RoboDK station: kr30 cnc 040719 6.rdk

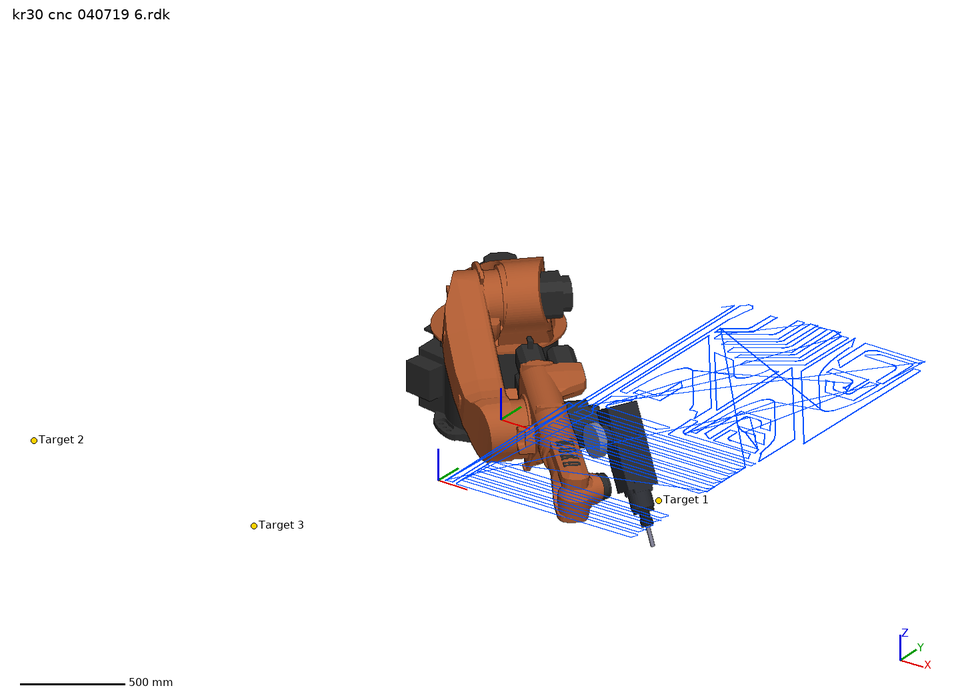
[picture v0: the station drawn from its stored meshes, robots at their saved joint values, targets as dots, program paths as lines]
Station kr30 cnc 040719 6. Poses are relative to the parent item; angles as X-Y-Z fixed-axis rotations.
  - frame KUKA KR 30 HA Base at (0, 0, 0) mm
    - robot KUKA KR 30 HA: 6 axes, payload 30 kg, reach 2033 mm, repeatability 0.05 mm, weight 665 kg
        modified DH rows (alpha deg, a mm, theta deg, d mm): 0, 0, 0, 815; -90, 350, 0, 0; 0, 850, -90, 0; -90, 145, 0, 820; 90, 0, 0, 0; -90, 0, 180, 170
        joint limits [-185, -135, -120, -350, -119, -350] to [185, 35, 158, 350, 119, 350]; home [0, -90, 90, 0, 0, 0]; saved at [44.88, 20.858, -14.182, 92.407, -109.74, -52.906]
      - tool 1/2" End Mill TCP, TCP at (337.71, -2.2, 160.57) mm, size 692.9 x 170 x 256 mm
    - frame Reference Rhino at (451.13, -1162.89, 269.68) mm
      - target Target 1 (Cartesian target) at (994.45, 406.4, 10) mm, rotated rx 0 ry 90 rz -60.43 deg; joints [16.304, -19.243, 71.371, -50.859, -63.853, 28.433] of KUKA KR 30 HA
      - target Target 2 (Cartesian target) at (-1810.84, -765.32, 10.08) mm, rotated rx 49.23 ry 89.99 rz -110.09 deg; joints [109.009, -5.295, 40.673, -64.339, -58.629, 47.297] of KUKA KR 30 HA
      - target Target 3 (Cartesian target) at (-425.52, -920.6, 10.08) mm, rotated rx 49.23 ry 89.99 rz -69.31 deg; joints [71.775, -8.447, 47.414, -59.408, -57.827, 42.008] of KUKA KR 30 HA
      - object RhinoPart at (0, 0, 0) mm
  - machining project RhinoPart Settings: C:/Users/Julian Ramirez.DESKTOP-JVDE542/Desktop/ELMER SHEET 1 TEST 3.nc | rotX(0) | rotY(270)*rotX(-65)
  - object box at (500, 500, 500) mm, size 250 x 250 x 250 mm, geometry from box.sld
  - program RhinoPart (634 instructions, listed below)
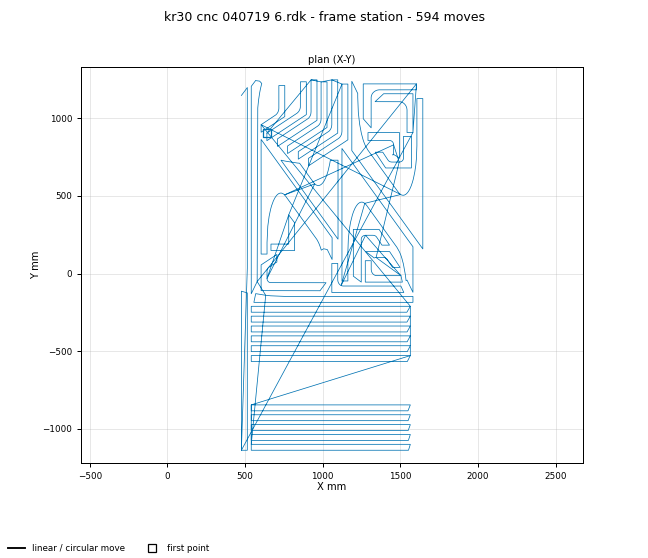
[picture p0: tool path of kr30 cnc 040719 6.rdk in frame station, 594 of 594 moves have a stored position in this frame; points joined in program order, loops and branches not executed]

--- program RhinoPart (robot KUKA KR 30 HA) ---
  Smooth(1)
  Set Ref.: Reference Rhino
  Set Tool: 1/2" End Mill TCP
  Show 1/2" End Mill TCP
  Set speed (2000.0 mm/s)
  MoveJ 1 to (189.6, 2067.69, 0) mm, rotated rx 0 ry 90 rz 65 deg; joints [-50.535, -45.887, 156.75, 15.433, -110.173, 5.438]
  MoveL 2 to (189.6, 2067.69, 0) mm, rotated rx 0 ry 90 rz 65 deg; joints [-50.535, -45.887, 156.75, 15.433, -110.173, 5.438]
  MoveL 3 to (189.6, 2067.69, 0) mm, rotated rx 0 ry 90 rz 65 deg; joints [-50.535, -45.887, 156.75, 15.433, -110.173, 5.438]
  Set speed (60.0 mm/s)
  MoveL 4 to (189.6, 2019.15, 0) mm, rotated rx 90 ry 80 rz 155 deg; joints [-43.975, -44.854, 157.735, 22.646, -111.28, -1.39]
  MoveL 5 to (443.6, 2187.03, 0) mm, rotated rx 0 ry 90 rz 65 deg; joints [-43.932, -46.602, 138.926, 21.084, -92.169, 0.836]
  MoveL 6 to (443.6, 2398.44, 0) mm, rotated rx 0 ry 90 rz 65 deg; joints [-51.209, -43.939, 127.221, 13.883, -83.477, -1.608]
  MoveL 7 to (405.5, 2398.44, 0) mm, rotated rx 0 ry 90 rz 65 deg; joints [-52.653, -44.436, 129.033, 12.401, -84.722, -1.159]
  MoveL 8 to (405.5, 2241.51, 0) mm, rotated rx 0 ry 90 rz 65 deg; joints [-47.49, -46.452, 138.026, 17.516, -91.501, 0.474]
  MoveL 9 to (405.1, 2234.61, 0) mm, rotated rx 0 ry 90 rz 65 deg; joints [-47.252, -46.518, 138.415, 17.757, -91.807, 0.578]
  MoveL 10 to (403.91, 2227.8, 0) mm, rotated rx 0 ry 90 rz 65 deg; joints [-47.047, -46.587, 138.835, 17.966, -92.138, 0.693]
  MoveL 11 to (401.94, 2221.18, 0) mm, rotated rx 0 ry 90 rz 65 deg; joints [-46.878, -46.658, 139.282, 18.139, -92.494, 0.817]
  MoveL 12 to (399.2, 2214.83, 0) mm, rotated rx 0 ry 90 rz 65 deg; joints [-46.749, -46.729, 139.751, 18.275, -92.87, 0.947]
  MoveL 13 to (395.69, 2208.84, 0) mm, rotated rx 0 ry 90 rz 65 deg; joints [-46.662, -46.8, 140.238, 18.369, -93.264, 1.083]
  MoveL 14 to (391.47, 2203.34, 0) mm, rotated rx 0 ry 90 rz 65 deg; joints [-46.623, -46.867, 140.732, 18.416, -93.667, 1.22]
  MoveL 15 to (386.58, 2198.44, 0) mm, rotated rx 0 ry 90 rz 65 deg; joints [-46.634, -46.931, 141.227, 18.415, -94.076, 1.356]
  MoveL 16 to (383.89, 2196.24, 0) mm, rotated rx 0 ry 90 rz 65 deg; joints [-46.659, -46.962, 141.472, 18.394, -94.281, 1.422]
  MoveL 17 to (381.06, 2194.23, 0) mm, rotated rx 0 ry 90 rz 65 deg; joints [-46.697, -46.991, 141.716, 18.361, -94.486, 1.487]
  MoveL 18 to (189.6, 2067.69, 0) mm, rotated rx 0 ry 90 rz 65 deg; joints [-50.535, -45.887, 156.75, 15.433, -110.173, 5.438]
  MoveL 19 to (474.07, 2410.87, 0) mm, rotated rx 0 ry 90 rz 65 deg; joints [-50.466, -43.286, 124.966, 14.682, -81.949, -2.102]
  Set speed (60.0 mm/s)
  MoveL 20 to (512.17, 2410.87, 0) mm, rotated rx 0 ry 90 rz 65 deg; joints [-49.125, -42.694, 123.02, 16.093, -80.698, -2.67]
  MoveL 21 to (512.17, 2150.2, 0) mm, rotated rx 0 ry 90 rz 65 deg; joints [-39.968, -46.268, 137.006, 25.034, -90.668, 0.312]
  MoveL 22 to (258.17, 1982.32, 0) mm, rotated rx 0 ry 90 rz 65 deg; joints [-42.535, -45.52, 157.698, 24.062, -110.416, 8.854]
  MoveL 23 to (258.17, 2030.85, 0) mm, rotated rx 0 ry 90 rz 65 deg; joints [-45.085, -46.283, 155.538, 20.995, -108.063, 6.786]
  MoveL 24 to (449.63, 2157.39, 0) mm, rotated rx 0 ry 90 rz 65 deg; joints [-42.511, -46.776, 140.073, 22.522, -93.046, 1.262]
  MoveL 25 to (455.15, 2161.61, 0) mm, rotated rx 0 ry 90 rz 65 deg; joints [-42.477, -46.703, 139.574, 22.548, -92.652, 1.101]
  MoveL 26 to (460.04, 2166.51, 0) mm, rotated rx 0 ry 90 rz 65 deg; joints [-42.494, -46.625, 139.075, 22.524, -92.263, 0.938]
  MoveL 27 to (464.26, 2172, 0) mm, rotated rx 0 ry 90 rz 65 deg; joints [-42.56, -46.545, 138.581, 22.453, -91.882, 0.777]
  MoveL 28 to (467.77, 2178, 0) mm, rotated rx 0 ry 90 rz 65 deg; joints [-42.67, -46.464, 138.099, 22.338, -91.512, 0.621]
  MoveL 29 to (470.51, 2184.35, 0) mm, rotated rx 0 ry 90 rz 65 deg; joints [-42.822, -46.384, 137.638, 22.183, -91.162, 0.474]
  MoveL 30 to (472.48, 2190.97, 0) mm, rotated rx 0 ry 90 rz 65 deg; joints [-43.01, -46.305, 137.204, 21.992, -90.834, 0.337]
  MoveL 31 to (474.07, 2204.68, 0) mm, rotated rx 0 ry 90 rz 65 deg; joints [-43.485, -46.159, 136.432, 21.516, -90.253, 0.1]
  MoveL 32 to (474.07, 2410.87, 0) mm, rotated rx 0 ry 90 rz 65 deg; joints [-50.466, -43.286, 124.966, 14.682, -81.949, -2.102]
  MoveL 33 to (538.73, 2397.73, 0) mm, rotated rx 0 ry 90 rz 65 deg; joints [-47.823, -42.501, 122.4, 17.431, -80.354, -3.011]
  Set speed (60.0 mm/s)
  MoveL 34 to (538.73, 2158.69, 0) mm, rotated rx 0 ry 90 rz 65 deg; joints [-39.418, -45.892, 135.103, 25.584, -89.288, -0.341]
  MoveL 35 to (537.14, 2144.98, 0) mm, rotated rx 0 ry 90 rz 65 deg; joints [-38.913, -46.041, 135.833, 26.087, -89.813, -0.092]
  MoveL 36 to (535.17, 2138.36, 0) mm, rotated rx 0 ry 90 rz 65 deg; joints [-38.706, -46.124, 136.251, 26.294, -90.114, 0.056]
  MoveL 37 to (532.43, 2132.01, 0) mm, rotated rx 0 ry 90 rz 65 deg; joints [-38.533, -46.211, 136.699, 26.467, -90.437, 0.218]
  MoveL 38 to (528.92, 2126.02, 0) mm, rotated rx 0 ry 90 rz 65 deg; joints [-38.399, -46.299, 137.173, 26.603, -90.782, 0.391]
  MoveL 39 to (524.7, 2120.53, 0) mm, rotated rx 0 ry 90 rz 65 deg; joints [-38.309, -46.388, 137.664, 26.697, -91.14, 0.573]
  MoveL 40 to (519.81, 2115.63, 0) mm, rotated rx 0 ry 90 rz 65 deg; joints [-38.264, -46.475, 138.164, 26.746, -91.508, 0.76]
  MoveL 41 to (514.29, 2111.41, 0) mm, rotated rx 0 ry 90 rz 65 deg; joints [-38.27, -46.56, 138.668, 26.745, -91.883, 0.949]
  MoveL 42 to (322.83, 1984.87, 0) mm, rotated rx 0 ry 90 rz 65 deg; joints [-39.614, -46.576, 154.441, 26.5, -106.091, 7.868]
  MoveL 43 to (322.83, 1936.34, 0) mm, rotated rx 0 ry 90 rz 65 deg; joints [-36.903, -46.012, 156.394, 29.663, -107.892, 9.925]
  MoveL 44 to (576.83, 2104.21, 0) mm, rotated rx 0 ry 90 rz 65 deg; joints [-35.947, -45.94, 135.336, 29.055, -89.472, -0.293]
  MoveL 45 to (576.83, 2397.73, 0) mm, rotated rx 0 ry 90 rz 65 deg; joints [-46.568, -41.834, 120.316, 18.784, -79.08, -3.686]
  MoveL 46 to (538.73, 2397.73, 0) mm, rotated rx 0 ry 90 rz 65 deg; joints [-47.823, -42.501, 122.4, 17.431, -80.354, -3.011]
  MoveL 47 to (607.72, 2410.87, 0) mm, rotated rx 0 ry 90 rz 65 deg; joints [-45.987, -40.997, 117.795, 19.491, -77.53, -4.37]
  Set speed (60.0 mm/s)
  MoveL 48 to (645.82, 2410.87, 0) mm, rotated rx 0 ry 90 rz 65 deg; joints [-44.821, -40.232, 115.572, 20.801, -76.258, -5.156]
  MoveL 49 to (645.82, 2068.09, 0) mm, rotated rx 0 ry 90 rz 65 deg; joints [-32.413, -45.334, 132.596, 32.617, -87.693, -1.476]
  MoveL 50 to (391.82, 1900.22, 0) mm, rotated rx 0 ry 90 rz 65 deg; joints [-32.027, -46.673, 154.021, 34.202, -104.486, 9.648]
  MoveL 51 to (391.82, 1948.75, 0) mm, rotated rx 0 ry 90 rz 65 deg; joints [-34.789, -47.001, 152.253, 31.112, -103.14, 7.812]
  MoveL 52 to (583.27, 2075.29, 0) mm, rotated rx 0 ry 90 rz 65 deg; joints [-34.508, -46.11, 136.177, 30.492, -90.058, 0.034]
  MoveL 53 to (588.8, 2079.51, 0) mm, rotated rx 0 ry 90 rz 65 deg; joints [-34.526, -46.008, 135.666, 30.474, -89.706, -0.173]
  MoveL 54 to (593.69, 2084.41, 0) mm, rotated rx 0 ry 90 rz 65 deg; joints [-34.592, -45.905, 135.164, 30.41, -89.361, -0.375]
  MoveL 55 to (597.91, 2089.9, 0) mm, rotated rx 0 ry 90 rz 65 deg; joints [-34.703, -45.802, 134.676, 30.302, -89.028, -0.568]
  MoveL 56 to (601.42, 2095.89, 0) mm, rotated rx 0 ry 90 rz 65 deg; joints [-34.854, -45.7, 134.208, 30.155, -88.709, -0.75]
  MoveL 57 to (604.16, 2102.24, 0) mm, rotated rx 0 ry 90 rz 65 deg; joints [-35.041, -45.603, 133.769, 29.972, -88.411, -0.916]
  MoveL 58 to (606.13, 2108.87, 0) mm, rotated rx 0 ry 90 rz 65 deg; joints [-35.26, -45.512, 133.364, 29.757, -88.135, -1.066]
  MoveL 59 to (607.72, 2122.58, 0) mm, rotated rx 0 ry 90 rz 65 deg; joints [-35.781, -45.352, 132.671, 29.246, -87.661, -1.309]
  MoveL 60 to (607.72, 2410.87, 0) mm, rotated rx 0 ry 90 rz 65 deg; joints [-45.987, -40.997, 117.795, 19.491, -77.53, -4.37]
  MoveL 61 to (673.1, 2383.75, 0) mm, rotated rx 0 ry 90 rz 65 deg; joints [-43.185, -40.209, 115.506, 22.481, -76.371, -5.569]
  Set speed (60.0 mm/s)
  MoveL 62 to (673.1, 2079.03, 0) mm, rotated rx 0 ry 90 rz 65 deg; joints [-32.147, -44.797, 130.411, 32.93, -86.317, -2.383]
  MoveL 63 to (671.52, 2065.32, 0) mm, rotated rx 0 ry 90 rz 65 deg; joints [-31.612, -44.962, 131.063, 33.449, -86.745, -2.148]
  MoveL 64 to (669.55, 2058.7, 0) mm, rotated rx 0 ry 90 rz 65 deg; joints [-31.381, -45.058, 131.452, 33.671, -86.997, -1.999]
  MoveL 65 to (666.8, 2052.35, 0) mm, rotated rx 0 ry 90 rz 65 deg; joints [-31.181, -45.163, 131.878, 33.863, -87.272, -1.83]
  MoveL 66 to (663.29, 2046.36, 0) mm, rotated rx 0 ry 90 rz 65 deg; joints [-31.014, -45.273, 132.337, 34.021, -87.566, -1.642]
  MoveL 67 to (659.07, 2040.86, 0) mm, rotated rx 0 ry 90 rz 65 deg; joints [-30.885, -45.387, 132.821, 34.141, -87.876, -1.44]
  MoveL 68 to (654.18, 2035.96, 0) mm, rotated rx 0 ry 90 rz 65 deg; joints [-30.799, -45.503, 133.323, 34.221, -88.198, -1.225]
  MoveL 69 to (648.66, 2031.74, 0) mm, rotated rx 0 ry 90 rz 65 deg; joints [-30.758, -45.619, 133.839, 34.255, -88.528, -1.002]
  MoveL 70 to (457.2, 1905.21, 0) mm, rotated rx 0 ry 90 rz 65 deg; joints [-30.057, -47.242, 150.114, 35.63, -100.522, 7.457]
  MoveL 71 to (457.2, 1856.67, 0) mm, rotated rx 0 ry 90 rz 65 deg; joints [-27.266, -47.081, 151.68, 38.648, -101.498, 9.056]
  MoveL 72 to (711.2, 2024.55, 0) mm, rotated rx 0 ry 90 rz 65 deg; joints [-28.881, -44.696, 130.018, 36.21, -86.223, -2.761]
  MoveL 73 to (711.2, 2383.75, 0) mm, rotated rx 0 ry 90 rz 65 deg; joints [-42.099, -39.37, 113.138, 23.748, -75.078, -6.464]
  MoveL 74 to (673.1, 2383.75, 0) mm, rotated rx 0 ry 90 rz 65 deg; joints [-43.185, -40.209, 115.506, 22.481, -76.371, -5.569]
  MoveL 75 to (330.2, 1541.24, 0) mm, rotated rx 90 ry 60 rz 155 deg; joints [-0.592, -40.922, 154.796, 66.348, -100.068, -8.239]
  Set speed (60.0 mm/s)
  MoveL 76 to (365.54, 1493.75, 0) mm, rotated rx 90 ry 70 rz 155 deg; joints [1.226, -43.408, 156.452, 67.934, -99.079, 1.27]
  MoveL 77 to (368.3, 1490.21, 0) mm, rotated rx 90 ry 70 rz 155 deg; joints [1.481, -43.485, 156.273, 68.137, -98.891, 1.067]
  MoveL 78 to (368.3, 1311.73, 0) mm, rotated rx 90 ry 70 rz 155 deg; joints [14.248, -44.077, 154.711, 79.923, -93.77, 0.302]
  MoveL 79 to (215.9, 1311.73, 0) mm, rotated rx 90 ry 50 rz 155 deg; joints [18.503, -36.104, 155.403, 84.328, -93.174, -10.858]
  MoveL 80 to (215.9, 1353.22, 0) mm, rotated rx 90 ry 50 rz 155 deg; joints [15.495, -35.61, 156.111, 81.791, -94.808, -9.844]
  MoveL 81 to (330.2, 1353.22, 0) mm, rotated rx 90 ry 70 rz 155 deg; joints [11.925, -42.84, 157.646, 78.096, -95.446, 4.238]
  MoveL 82 to (330.2, 1541.24, 0) mm, rotated rx 90 ry 60 rz 155 deg; joints [-0.592, -40.922, 154.796, 66.348, -100.068, -8.239]
  MoveL 83 to (190.5, 1131.98, 0) mm, rotated rx 90 ry 60 rz 155 deg; joints [31.549, -40.102, 156.424, 95.875, -87.101, -3.827]
  Set speed (60.0 mm/s)
  MoveL 84 to (190.5, 1180.23, 0) mm, rotated rx 90 ry 60 rz 155 deg; joints [28.374, -39.204, 157.878, 92.961, -88.382, -1.368]
  MoveL 85 to (191.3, 1187.11, 0) mm, rotated rx 90 ry 50 rz 155 deg; joints [27.699, -37.052, 153.838, 92.41, -88.784, -13.24]
  MoveL 86 to (192.29, 1190.42, 0) mm, rotated rx 90 ry 50 rz 155 deg; joints [27.453, -37.03, 153.877, 92.188, -88.893, -13.174]
  MoveL 87 to (193.65, 1193.58, 0) mm, rotated rx 90 ry 50 rz 155 deg; joints [27.202, -37.022, 153.892, 91.965, -89.005, -13.148]
  MoveL 88 to (195.39, 1196.56, 0) mm, rotated rx 90 ry 50 rz 155 deg; joints [26.952, -37.029, 153.88, 91.742, -89.118, -13.162]
  MoveL 89 to (197.49, 1199.29, 0) mm, rotated rx 90 ry 50 rz 155 deg; joints [26.706, -37.05, 153.842, 91.523, -89.231, -13.218]
  MoveL 90 to (199.93, 1201.75, 0) mm, rotated rx 90 ry 60 rz 155 deg; joints [26.563, -39.14, 157.97, 91.369, -89.246, -1.179]
  MoveL 91 to (202.72, 1203.88, 0) mm, rotated rx 90 ry 60 rz 155 deg; joints [26.32, -39.203, 157.878, 91.158, -89.367, -1.332]
  MoveL 92 to (254, 1237.77, 0) mm, rotated rx 90 ry 60 rz 155 deg; joints [22.391, -40.388, 155.895, 87.645, -91.123, -4.516]
  MoveL 93 to (254, 1286.3, 0) mm, rotated rx 90 ry 60 rz 155 deg; joints [18.997, -39.802, 156.941, 84.654, -92.734, -2.989]
  MoveL 94 to (152.4, 1219.15, 0) mm, rotated rx 90 ry 50 rz 155 deg; joints [26.902, -35.139, 156.733, 91.62, -89.004, -8.421]
  MoveL 95 to (152.4, 1053.37, 0) mm, rotated rx 90 ry 60 rz 155 deg; joints [37.947, -40.542, 155.596, 101.764, -84.556, -5.508]
  MoveL 96 to (520.7, 1053.37, 0) mm, rotated rx 0 ry 90 rz 65 deg; joints [26.184, -47.344, 147.433, 91.166, -89.793, 10.087]
  MoveL 97 to (523.39, 1053.29, 0) mm, rotated rx 0 ry 90 rz 65 deg; joints [26.115, -47.344, 147.265, 91.098, -89.808, 9.919]
  MoveL 98 to (526.09, 1053.06, 0) mm, rotated rx 0 ry 90 rz 65 deg; joints [26.055, -47.343, 147.091, 91.04, -89.821, 9.746]
  MoveL 99 to (528.75, 1052.67, 0) mm, rotated rx 0 ry 90 rz 65 deg; joints [26.005, -47.341, 146.914, 90.991, -89.833, 9.571]
  MoveL 100 to (531.38, 1052.13, 0) mm, rotated rx 0 ry 90 rz 65 deg; joints [25.964, -47.339, 146.734, 90.951, -89.843, 9.394]
  MoveL 101 to (570.41, 1104.33, 0) mm, rotated rx 0 ry 90 rz 65 deg; joints [22.098, -47.312, 145.737, 87.13, -90.425, 8.414]
  MoveL 102 to (215.9, 1104.33, 0) mm, rotated rx 90 ry 60 rz 155 deg; joints [32.283, -41.184, 154.189, 96.709, -87.16, -7.162]
  MoveL 103 to (210.71, 1104.91, 0) mm, rotated rx 90 ry 60 rz 155 deg; joints [32.446, -41.06, 154.482, 96.839, -87.047, -6.755]
  MoveL 104 to (208.23, 1105.62, 0) mm, rotated rx 90 ry 60 rz 155 deg; joints [32.499, -40.993, 154.636, 96.876, -87, -6.538]
  MoveL 105 to (205.85, 1106.58, 0) mm, rotated rx 90 ry 60 rz 155 deg; joints [32.532, -40.923, 154.793, 96.895, -86.959, -6.313]
  MoveL 106 to (203.58, 1107.8, 0) mm, rotated rx 90 ry 60 rz 155 deg; joints [32.547, -40.851, 154.953, 96.895, -86.926, -6.083]
  MoveL 107 to (201.44, 1109.25, 0) mm, rotated rx 90 ry 60 rz 155 deg; joints [32.542, -40.776, 155.113, 96.878, -86.9, -5.85]
  MoveL 108 to (199.45, 1110.91, 0) mm, rotated rx 90 ry 60 rz 155 deg; joints [32.517, -40.701, 155.272, 96.843, -86.881, -5.615]
  MoveL 109 to (197.61, 1112.79, 0) mm, rotated rx 90 ry 60 rz 155 deg; joints [32.474, -40.624, 155.43, 96.791, -86.872, -5.38]
  MoveL 110 to (195.97, 1114.84, 0) mm, rotated rx 90 ry 60 rz 155 deg; joints [32.412, -40.548, 155.583, 96.722, -86.871, -5.148]
  MoveL 111 to (194.53, 1117.03, 0) mm, rotated rx 90 ry 60 rz 155 deg; joints [32.332, -40.474, 155.73, 96.638, -86.879, -4.925]
  MoveL 112 to (192.31, 1121.74, 0) mm, rotated rx 90 ry 60 rz 155 deg; joints [32.126, -40.333, 156, 96.429, -86.92, -4.507]
  MoveL 113 to (190.96, 1126.77, 0) mm, rotated rx 90 ry 60 rz 155 deg; joints [31.862, -40.208, 156.233, 96.171, -86.995, -4.137]
  MoveL 114 to (190.5, 1131.98, 0) mm, rotated rx 90 ry 60 rz 155 deg; joints [31.549, -40.102, 156.424, 95.875, -87.101, -3.827]
  MoveL 115 to (497.79, 1740.88, 0) mm, rotated rx 90 ry 70 rz 155 deg; joints [-14.18, -45.425, 145.857, 51.287, -96.568, -11.878]
  Set speed (60.0 mm/s)
  MoveL 116 to (502.27, 1737.01, 0) mm, rotated rx 0 ry 90 rz 65 deg; joints [-18.744, -47.033, 152.033, 47.247, -100.309, 10.956]
  MoveL 117 to (506.69, 1734.05, 0) mm, rotated rx 0 ry 90 rz 65 deg; joints [-18.463, -47.063, 151.817, 47.495, -100.089, 10.821]
  MoveL 118 to (511.04, 1731.95, 0) mm, rotated rx 0 ry 90 rz 65 deg; joints [-18.239, -47.093, 151.585, 47.684, -99.871, 10.664]
  MoveL 119 to (515.31, 1730.65, 0) mm, rotated rx 0 ry 90 rz 65 deg; joints [-18.069, -47.123, 151.34, 47.819, -99.655, 10.486]
  MoveL 120 to (519.5, 1730.11, 0) mm, rotated rx 0 ry 90 rz 65 deg; joints [-17.95, -47.152, 151.084, 47.902, -99.442, 10.291]
  MoveL 121 to (523.61, 1730.27, 0) mm, rotated rx 0 ry 90 rz 65 deg; joints [-17.878, -47.18, 150.818, 47.939, -99.232, 10.082]
  MoveL 122 to (527.62, 1731.09, 0) mm, rotated rx 0 ry 90 rz 65 deg; joints [-17.848, -47.206, 150.544, 47.932, -99.026, 9.861]
  MoveL 123 to (531.52, 1732.52, 0) mm, rotated rx 0 ry 90 rz 65 deg; joints [-17.859, -47.23, 150.264, 47.886, -98.824, 9.631]
  MoveL 124 to (535.31, 1734.5, 0) mm, rotated rx 0 ry 90 rz 65 deg; joints [-17.906, -47.252, 149.979, 47.804, -98.626, 9.394]
  MoveL 125 to (538.98, 1736.99, 0) mm, rotated rx 0 ry 90 rz 65 deg; joints [-17.985, -47.272, 149.691, 47.691, -98.432, 9.151]
  MoveL 126 to (542.53, 1739.94, 0) mm, rotated rx 0 ry 90 rz 65 deg; joints [-18.094, -47.289, 149.4, 47.548, -98.241, 8.906]
  MoveL 127 to (545.93, 1743.29, 0) mm, rotated rx 0 ry 90 rz 65 deg; joints [-18.23, -47.304, 149.109, 47.381, -98.055, 8.659]
  MoveL 128 to (552.31, 1751, 0) mm, rotated rx 0 ry 90 rz 65 deg; joints [-18.566, -47.327, 148.531, 46.984, -97.696, 8.168]
  MoveL 129 to (557.85, 1759.34, 0) mm, rotated rx 0 ry 90 rz 65 deg; joints [-18.95, -47.339, 147.988, 46.548, -97.369, 7.71]
  MoveL 130 to (562.91, 1768.41, 0) mm, rotated rx 0 ry 90 rz 65 deg; joints [-19.379, -47.344, 147.456, 46.069, -97.053, 7.264]
  MoveL 131 to (567.51, 1777.97, 0) mm, rotated rx 0 ry 90 rz 65 deg; joints [-19.839, -47.342, 146.936, 45.564, -96.749, 6.835]
  MoveL 132 to (576.13, 1799.75, 0) mm, rotated rx 0 ry 90 rz 65 deg; joints [-20.901, -47.316, 145.852, 44.418, -96.119, 5.963]
  MoveL 133 to (584.02, 1825.23, 0) mm, rotated rx 0 ry 90 rz 65 deg; joints [-22.148, -47.259, 144.689, 43.093, -95.44, 5.068]
  MoveL 134 to (593.39, 1865.46, 0) mm, rotated rx 0 ry 90 rz 65 deg; joints [-24.102, -47.124, 142.972, 41.046, -94.417, 3.836]
  MoveL 135 to (598.13, 1892.37, 0) mm, rotated rx 0 ry 90 rz 65 deg; joints [-25.393, -47.008, 141.868, 39.709, -93.742, 3.102]
  MoveL 136 to (609.6, 1893.44, 0) mm, rotated rx 0 ry 90 rz 65 deg; joints [-25.17, -46.915, 141.096, 39.905, -93.21, 2.681]
  MoveL 137 to (647.7, 1893.44, 0) mm, rotated rx 0 ry 90 rz 65 deg; joints [-24.286, -46.549, 138.606, 40.733, -91.558, 1.341]
  MoveL 138 to (647.7, 1384.85, 0) mm, rotated rx 0 ry 90 rz 65 deg; joints [4.583, -47.277, 144.998, 69.753, -92.686, 7.241]
  MoveL 139 to (280.37, 1893.44, 0) mm, rotated rx 90 ry 70 rz 155 deg; joints [-28.872, -43.751, 155.615, 38.186, -107.505, -6.69]
  MoveL 140 to (309.91, 1887.14, 0) mm, rotated rx 90 ry 80 rz 155 deg; joints [-30.792, -45.262, 156.747, 36.15, -107.632, 2.478]
  MoveL 141 to (385.37, 1875.31, 0) mm, rotated rx 0 ry 90 rz 65 deg; joints [-30.773, -46.371, 155.229, 35.711, -105.5, 10.875]
  MoveL 142 to (400.34, 1873.88, 0) mm, rotated rx 0 ry 90 rz 65 deg; joints [-30.153, -46.577, 154.434, 36.184, -104.575, 10.43]
  MoveL 143 to (488.7, 1751.54, 0) mm, rotated rx 0 ry 90 rz 65 deg; joints [-19.967, -46.952, 152.565, 46.11, -100.964, 11.184]
  MoveL 144 to (493.27, 1745.7, 0) mm, rotated rx 0 ry 90 rz 65 deg; joints [-19.493, -46.977, 152.41, 46.558, -100.748, 11.141]
  MoveL 145 to (497.79, 1740.88, 0) mm, rotated rx 0 ry 90 rz 65 deg; joints [-19.086, -47.004, 152.232, 46.936, -100.529, 11.063]
  MoveL 146 to (303.35, 1670.14, 0) mm, rotated rx 90 ry 60 rz 155 deg; joints [-10.146, -40.486, 155.706, 57.507, -104.199, -8.936]
  Set speed (60.0 mm/s)
  MoveL 147 to (307.39, 1665.7, 0) mm, rotated rx 90 ry 60 rz 155 deg; joints [-9.773, -40.585, 155.508, 57.803, -103.906, -9.109]
  MoveL 148 to (311.4, 1660.54, 0) mm, rotated rx 90 ry 60 rz 155 deg; joints [-9.352, -40.679, 155.317, 58.149, -103.606, -9.261]
  MoveL 149 to (511.79, 1382.48, 0) mm, rotated rx 0 ry 90 rz 65 deg; joints [5.501, -46.642, 154.16, 71.341, -95.767, 16.57]
  MoveL 150 to (516.77, 1373.81, 0) mm, rotated rx 0 ry 90 rz 65 deg; joints [6.063, -46.726, 153.777, 71.84, -95.46, 16.178]
  MoveL 151 to (521.42, 1364.56, 0) mm, rotated rx 0 ry 90 rz 65 deg; joints [6.659, -46.802, 153.405, 72.375, -95.158, 15.802]
  MoveL 152 to (525.76, 1354.87, 0) mm, rotated rx 0 ry 90 rz 65 deg; joints [7.28, -46.87, 153.042, 72.94, -94.863, 15.442]
  MoveL 153 to (533.5, 1334.64, 0) mm, rotated rx 0 ry 90 rz 65 deg; joints [8.563, -46.987, 152.348, 74.12, -94.299, 14.762]
  MoveL 154 to (540.04, 1314.08, 0) mm, rotated rx 0 ry 90 rz 65 deg; joints [9.849, -47.079, 151.698, 75.318, -93.782, 14.132]
  MoveL 155 to (555.23, 1322.96, 0) mm, rotated rx 0 ry 90 rz 65 deg; joints [9.107, -47.183, 150.792, 74.532, -93.694, 13.107]
  MoveL 156 to (561.07, 1321.73, 0) mm, rotated rx 0 ry 90 rz 65 deg; joints [9.126, -47.22, 150.39, 74.523, -93.573, 12.684]
  MoveL 157 to (578.58, 1317.86, 0) mm, rotated rx 0 ry 90 rz 65 deg; joints [9.192, -47.301, 149.177, 74.514, -93.214, 11.439]
  MoveL 158 to (609.6, 1253.88, 0) mm, rotated rx 0 ry 90 rz 65 deg; joints [12.734, -47.329, 146.25, 77.878, -91.888, 8.721]
  MoveL 159 to (609.6, 1394.22, 0) mm, rotated rx 0 ry 90 rz 65 deg; joints [4.191, -47.343, 147.678, 69.501, -93.654, 9.675]
  MoveL 160 to (152.4, 2027.23, 0) mm, rotated rx 90 ry 60 rz 155 deg; joints [-38.777, -40.811, 155.04, 28.375, -111.602, -18.753]
  MoveL 161 to (152.4, 1288.87, 0) mm, rotated rx 90 ry 20 rz 155 deg; joints [22.268, -23.754, 146.138, 87.693, -91.463, -37.646]
  MoveL 162 to (190.5, 1288.87, 0) mm, rotated rx 90 ry 50 rz 155 deg; joints [20.788, -35.434, 156.349, 86.385, -92.162, -9.154]
  MoveL 163 to (190.5, 1362.91, 0) mm, rotated rx 90 ry 50 rz 155 deg; joints [15.292, -34.367, 157.659, 81.862, -95.311, -7.087]
  MoveL 164 to (195.47, 1468.11, 0) mm, rotated rx 90 ry 40 rz 155 deg; joints [7.932, -30.96, 154.459, 75.639, -99.323, -17.678]
  MoveL 165 to (203.82, 1530.87, 0) mm, rotated rx 90 ry 40 rz 155 deg; joints [3.087, -31.064, 154.333, 71.41, -101.813, -18.672]
  MoveL 166 to (213.36, 1576.46, 0) mm, rotated rx 90 ry 50 rz 155 deg; joints [-1.825, -34.249, 157.792, 67.146, -104.439, -9.39]
  MoveL 167 to (219.68, 1599.23, 0) mm, rotated rx 90 ry 50 rz 155 deg; joints [-3.601, -34.614, 157.375, 65.368, -105.013, -10.535]
  MoveL 168 to (227.14, 1620.99, 0) mm, rotated rx 90 ry 50 rz 155 deg; joints [-5.253, -35.042, 156.855, 63.636, -105.402, -11.815]
  MoveL 169 to (231.16, 1630.88, 0) mm, rotated rx 90 ry 50 rz 155 deg; joints [-5.985, -35.266, 156.57, 62.838, -105.515, -12.466]
  MoveL 170 to (235.75, 1640.83, 0) mm, rotated rx 90 ry 50 rz 155 deg; joints [-6.707, -35.513, 156.243, 62.03, -105.579, -13.173]
  MoveL 171 to (240.92, 1650.5, 0) mm, rotated rx 90 ry 50 rz 155 deg; joints [-7.391, -35.779, 155.877, 61.239, -105.583, -13.921]
  MoveL 172 to (246.67, 1659.52, 0) mm, rotated rx 90 ry 50 rz 155 deg; joints [-8.009, -36.057, 155.473, 60.495, -105.52, -14.694]
  MoveL 173 to (250.51, 1664.62, 0) mm, rotated rx 90 ry 50 rz 155 deg; joints [-8.347, -36.233, 155.207, 60.071, -105.443, -15.177]
  MoveL 174 to (254.42, 1669.07, 0) mm, rotated rx 90 ry 50 rz 155 deg; joints [-8.633, -36.404, 154.94, 59.698, -105.343, -15.641]
  MoveL 175 to (258.37, 1672.87, 0) mm, rotated rx 90 ry 50 rz 155 deg; joints [-8.867, -36.568, 154.675, 59.375, -105.22, -16.084]
  MoveL 176 to (262.38, 1676.02, 0) mm, rotated rx 90 ry 50 rz 155 deg; joints [-9.05, -36.727, 154.41, 59.103, -105.078, -16.506]
  MoveL 177 to (266.41, 1678.5, 0) mm, rotated rx 90 ry 60 rz 155 deg; joints [-11.281, -39.247, 157.813, 57.19, -106.436, -6.304]
  MoveL 178 to (270.48, 1680.31, 0) mm, rotated rx 90 ry 60 rz 155 deg; joints [-11.356, -39.42, 157.553, 57.011, -106.232, -6.703]
  MoveL 179 to (274.58, 1681.45, 0) mm, rotated rx 90 ry 60 rz 155 deg; joints [-11.38, -39.582, 157.298, 56.887, -106.013, -7.073]
  MoveL 180 to (278.69, 1681.92, 0) mm, rotated rx 90 ry 60 rz 155 deg; joints [-11.353, -39.736, 157.049, 56.817, -105.783, -7.417]
  MoveL 181 to (282.81, 1681.7, 0) mm, rotated rx 90 ry 60 rz 155 deg; joints [-11.276, -39.881, 156.807, 56.801, -105.541, -7.733]
  MoveL 182 to (286.94, 1680.79, 0) mm, rotated rx 90 ry 60 rz 155 deg; joints [-11.148, -40.018, 156.572, 56.838, -105.29, -8.023]
  MoveL 183 to (291.06, 1679.18, 0) mm, rotated rx 90 ry 60 rz 155 deg; joints [-10.971, -40.146, 156.345, 56.927, -105.03, -8.287]
  MoveL 184 to (295.17, 1676.87, 0) mm, rotated rx 90 ry 60 rz 155 deg; joints [-10.745, -40.267, 156.125, 57.069, -104.761, -8.527]
  MoveL 185 to (299.27, 1673.86, 0) mm, rotated rx 90 ry 60 rz 155 deg; joints [-10.47, -40.38, 155.912, 57.263, -104.484, -8.743]
  MoveL 186 to (303.35, 1670.14, 0) mm, rotated rx 90 ry 60 rz 155 deg; joints [-10.146, -40.486, 155.706, 57.507, -104.199, -8.936]
  MoveL 187 to (1005.83, 1992.41, 0) mm, rotated rx 0 ry 90 rz 65 deg; joints [-21.979, -38.015, 109.438, 44.552, -76.532, -12.914]
  Set speed (60.0 mm/s)
  MoveL 188 to (1005.72, 1995.03, 0) mm, rotated rx 0 ry 90 rz 65 deg; joints [-22.079, -37.986, 109.361, 44.46, -76.475, -12.926]
  MoveL 189 to (1005.38, 1997.62, 0) mm, rotated rx 0 ry 90 rz 65 deg; joints [-22.181, -37.964, 109.303, 44.364, -76.426, -12.928]
  MoveL 190 to (1004.81, 2000.17, 0) mm, rotated rx 0 ry 90 rz 65 deg; joints [-22.285, -37.95, 109.264, 44.264, -76.386, -12.921]
  MoveL 191 to (1004.02, 2002.66, 0) mm, rotated rx 0 ry 90 rz 65 deg; joints [-22.39, -37.943, 109.245, 44.161, -76.354, -12.905]
  MoveL 192 to (1003.02, 2005.06, 0) mm, rotated rx 0 ry 90 rz 65 deg; joints [-22.495, -37.943, 109.246, 44.055, -76.331, -12.879]
  MoveL 193 to (1001.8, 2007.37, 0) mm, rotated rx 0 ry 90 rz 65 deg; joints [-22.6, -37.951, 109.268, 43.948, -76.317, -12.845]
  MoveL 194 to (1000.36, 2009.56, 0) mm, rotated rx 0 ry 90 rz 65 deg; joints [-22.703, -37.967, 109.31, 43.839, -76.313, -12.801]
  MoveL 195 to (998.72, 2011.61, 0) mm, rotated rx 0 ry 90 rz 65 deg; joints [-22.805, -37.991, 109.374, 43.73, -76.319, -12.749]
  MoveL 196 to (996.89, 2013.48, 0) mm, rotated rx 0 ry 90 rz 65 deg; joints [-22.904, -38.022, 109.458, 43.622, -76.336, -12.688]
  MoveL 197 to (994.89, 2015.15, 0) mm, rotated rx 0 ry 90 rz 65 deg; joints [-22.997, -38.061, 109.562, 43.518, -76.362, -12.62]
  MoveL 198 to (992.75, 2016.6, 0) mm, rotated rx 0 ry 90 rz 65 deg; joints [-23.085, -38.106, 109.684, 43.417, -76.399, -12.544]
  MoveL 199 to (990.48, 2017.81, 0) mm, rotated rx 0 ry 90 rz 65 deg; joints [-23.167, -38.159, 109.825, 43.32, -76.446, -12.463]
  MoveL 200 to (988.1, 2018.78, 0) mm, rotated rx 0 ry 90 rz 65 deg; joints [-23.241, -38.218, 109.983, 43.229, -76.502, -12.375]
  MoveL 201 to (985.62, 2019.49, 0) mm, rotated rx 0 ry 90 rz 65 deg; joints [-23.307, -38.282, 110.157, 43.145, -76.568, -12.283]
  MoveL 202 to (983.06, 2019.92, 0) mm, rotated rx 0 ry 90 rz 65 deg; joints [-23.364, -38.352, 110.347, 43.068, -76.643, -12.185]
  MoveL 203 to (980.43, 2020.07, 0) mm, rotated rx 0 ry 90 rz 65 deg; joints [-23.412, -38.428, 110.552, 42.999, -76.727, -12.084]
  MoveL 204 to (840.73, 2020.07, 0) mm, rotated rx 0 ry 90 rz 65 deg; joints [-25.901, -42.11, 121.168, 39.615, -81.529, -6.952]
  MoveL 205 to (840.73, 2071.02, 0) mm, rotated rx 0 ry 90 rz 65 deg; joints [-27.919, -41.5, 119.297, 37.713, -80.292, -7.429]
  MoveL 206 to (1043.93, 2071.02, 0) mm, rotated rx 0 ry 90 rz 65 deg; joints [-24.243, -35.75, 103.522, 42.955, -73.348, -14.938]
  MoveL 207 to (1043.93, 1907.58, 0) mm, rotated rx 0 ry 90 rz 65 deg; joints [-18.24, -37.797, 108.857, 48.348, -77.153, -14.036]
  MoveL 208 to (1015.37, 1924.76, 0) mm, rotated rx 0 ry 90 rz 65 deg; joints [-19.271, -38.497, 110.738, 47.126, -77.707, -12.916]
  MoveL 209 to (1005.83, 1930.45, 0) mm, rotated rx 0 ry 90 rz 65 deg; joints [-19.621, -38.723, 111.353, 46.715, -77.895, -12.552]
  MoveL 210 to (1000.11, 1926.67, 0) mm, rotated rx 0 ry 90 rz 65 deg; joints [-19.553, -38.932, 111.927, 46.726, -78.16, -12.294]
  MoveL 211 to (1001.43, 1928.6, 0) mm, rotated rx 0 ry 90 rz 65 deg; joints [-19.61, -38.873, 111.764, 46.686, -78.077, -12.36]
  MoveL 212 to (1002.59, 1930.63, 0) mm, rotated rx 0 ry 90 rz 65 deg; joints [-19.673, -38.817, 111.612, 46.638, -77.997, -12.419]
  MoveL 213 to (1003.57, 1932.75, 0) mm, rotated rx 0 ry 90 rz 65 deg; joints [-19.741, -38.766, 111.47, 46.584, -77.921, -12.471]
  MoveL 214 to (1004.38, 1934.94, 0) mm, rotated rx 0 ry 90 rz 65 deg; joints [-19.814, -38.718, 111.34, 46.523, -77.848, -12.517]
  MoveL 215 to (1005.01, 1937.19, 0) mm, rotated rx 0 ry 90 rz 65 deg; joints [-19.892, -38.675, 111.223, 46.457, -77.78, -12.556]
  MoveL 216 to (1005.47, 1939.49, 0) mm, rotated rx 0 ry 90 rz 65 deg; joints [-19.974, -38.637, 111.118, 46.385, -77.716, -12.588]
  MoveL 217 to (1005.83, 1944.16, 0) mm, rotated rx 0 ry 90 rz 65 deg; joints [-20.149, -38.575, 110.949, 46.228, -77.604, -12.629]
  MoveL 218 to (1005.83, 1992.41, 0) mm, rotated rx 0 ry 90 rz 65 deg; joints [-21.979, -38.015, 109.438, 44.552, -76.532, -12.914]
  MoveL 219 to (1041.7, 1881.48, 0) mm, rotated rx 0 ry 90 rz 65 deg; joints [-17.265, -38.128, 109.742, 49.225, -77.752, -13.819]
  Set speed (60.0 mm/s)
  MoveL 220 to (993.45, 1881.48, 0) mm, rotated rx 0 ry 90 rz 65 deg; joints [-17.864, -39.573, 113.704, 48.244, -79.28, -11.77]
  MoveL 221 to (986.57, 1882.28, 0) mm, rotated rx 0 ry 90 rz 65 deg; joints [-17.985, -39.763, 114.238, 48.076, -79.485, -11.487]
  MoveL 222 to (983.26, 1883.27, 0) mm, rotated rx 0 ry 90 rz 65 deg; joints [-18.067, -39.848, 114.478, 47.972, -79.572, -11.355]
  MoveL 223 to (980.1, 1884.64, 0) mm, rotated rx 0 ry 90 rz 65 deg; joints [-18.164, -39.925, 114.696, 47.857, -79.648, -11.231]
  MoveL 224 to (977.13, 1886.37, 0) mm, rotated rx 0 ry 90 rz 65 deg; joints [-18.273, -39.992, 114.888, 47.732, -79.71, -11.118]
  MoveL 225 to (974.39, 1888.47, 0) mm, rotated rx 0 ry 90 rz 65 deg; joints [-18.393, -40.05, 115.051, 47.597, -79.758, -11.017]
  MoveL 226 to (971.94, 1890.91, 0) mm, rotated rx 0 ry 90 rz 65 deg; joints [-18.524, -40.096, 115.181, 47.455, -79.791, -10.931]
  MoveL 227 to (969.81, 1893.7, 0) mm, rotated rx 0 ry 90 rz 65 deg; joints [-18.665, -40.129, 115.276, 47.306, -79.806, -10.86]
  MoveL 228 to (935.92, 1944.98, 0) mm, rotated rx 0 ry 90 rz 65 deg; joints [-21.215, -40.546, 116.477, 44.657, -79.892, -9.838]
  MoveL 229 to (887.38, 1944.98, 0) mm, rotated rx 0 ry 90 rz 65 deg; joints [-21.995, -41.791, 120.184, 43.596, -81.539, -7.975]
  MoveL 230 to (954.53, 1843.38, 0) mm, rotated rx 0 ry 90 rz 65 deg; joints [-16.808, -40.985, 117.762, 48.955, -81.228, -9.935]
  MoveL 231 to (1120.31, 1843.38, 0) mm, rotated rx 0 ry 90 rz 65 deg; joints [-14.952, -35.908, 103.927, 52.161, -76.092, -17.194]
  MoveL 232 to (1120.31, 2046.58, 0) mm, rotated rx 0 ry 90 rz 65 deg; joints [-22.253, -33.469, 97.812, 45.718, -71.46, -18.058]
  MoveL 233 to (1069.36, 2046.58, 0) mm, rotated rx 0 ry 90 rz 65 deg; joints [-22.991, -35.258, 102.273, 44.373, -73.133, -15.848]
  MoveL 234 to (1069.36, 1906.88, 0) mm, rotated rx 0 ry 90 rz 65 deg; joints [-17.899, -36.991, 106.729, 48.92, -76.365, -15.132]
  MoveL 235 to (1069.21, 1904.25, 0) mm, rotated rx 0 ry 90 rz 65 deg; joints [-17.802, -37.024, 106.814, 49.007, -76.424, -15.115]
  MoveL 236 to (1068.78, 1901.69, 0) mm, rotated rx 0 ry 90 rz 65 deg; joints [-17.711, -37.065, 106.921, 49.086, -76.492, -15.084]
  MoveL 237 to (1068.07, 1899.21, 0) mm, rotated rx 0 ry 90 rz 65 deg; joints [-17.626, -37.113, 107.048, 49.156, -76.565, -15.043]
  MoveL 238 to (1067.1, 1896.83, 0) mm, rotated rx 0 ry 90 rz 65 deg; joints [-17.547, -37.169, 107.195, 49.218, -76.645, -14.99]
  MoveL 239 to (1065.89, 1894.56, 0) mm, rotated rx 0 ry 90 rz 65 deg; joints [-17.476, -37.231, 107.359, 49.27, -76.73, -14.927]
  MoveL 240 to (1064.44, 1892.42, 0) mm, rotated rx 0 ry 90 rz 65 deg; joints [-17.412, -37.3, 107.539, 49.314, -76.819, -14.855]
  MoveL 241 to (1062.77, 1890.43, 0) mm, rotated rx 0 ry 90 rz 65 deg; joints [-17.356, -37.374, 107.734, 49.348, -76.912, -14.773]
  MoveL 242 to (1060.9, 1888.6, 0) mm, rotated rx 0 ry 90 rz 65 deg; joints [-17.308, -37.452, 107.941, 49.373, -77.008, -14.684]
  MoveL 243 to (1058.85, 1886.95, 0) mm, rotated rx 0 ry 90 rz 65 deg; joints [-17.27, -37.534, 108.158, 49.387, -77.106, -14.587]
  MoveL 244 to (1056.66, 1885.52, 0) mm, rotated rx 0 ry 90 rz 65 deg; joints [-17.241, -37.618, 108.38, 49.392, -77.203, -14.486]
  MoveL 245 to (1054.35, 1884.29, 0) mm, rotated rx 0 ry 90 rz 65 deg; joints [-17.222, -37.703, 108.607, 49.387, -77.3, -14.38]
  MoveL 246 to (1051.95, 1883.29, 0) mm, rotated rx 0 ry 90 rz 65 deg; joints [-17.212, -37.789, 108.836, 49.373, -77.395, -14.271]
  MoveL 247 to (1049.46, 1882.5, 0) mm, rotated rx 0 ry 90 rz 65 deg; joints [-17.211, -37.875, 109.065, 49.349, -77.489, -14.16]
  MoveL 248 to (1046.91, 1881.94, 0) mm, rotated rx 0 ry 90 rz 65 deg; joints [-17.22, -37.961, 109.294, 49.316, -77.58, -14.047]
  MoveL 249 to (1044.32, 1881.6, 0) mm, rotated rx 0 ry 90 rz 65 deg; joints [-17.238, -38.045, 109.52, 49.275, -77.668, -13.933]
  MoveL 250 to (1041.7, 1881.48, 0) mm, rotated rx 0 ry 90 rz 65 deg; joints [-17.265, -38.128, 109.742, 49.225, -77.752, -13.819]
  MoveL 251 to (892.95, 1266.65, 0) mm, rotated rx 0 ry 90 rz 65 deg; joints [9.208, -43.581, 125.97, 74.34, -87.934, -7.327]
  Set speed (60.0 mm/s)
  MoveL 252 to (889.54, 1266.46, 0) mm, rotated rx 0 ry 90 rz 65 deg; joints [9.243, -43.656, 126.229, 74.368, -87.988, -7.151]
  MoveL 253 to (886.2, 1265.88, 0) mm, rotated rx 0 ry 90 rz 65 deg; joints [9.295, -43.728, 126.48, 74.414, -88.043, -6.981]
  MoveL 254 to (882.94, 1264.93, 0) mm, rotated rx 0 ry 90 rz 65 deg; joints [9.364, -43.796, 126.718, 74.478, -88.097, -6.819]
  MoveL 255 to (879.82, 1263.61, 0) mm, rotated rx 0 ry 90 rz 65 deg; joints [9.451, -43.859, 126.94, 74.558, -88.149, -6.668]
  MoveL 256 to (876.88, 1266.65, 0) mm, rotated rx 0 ry 90 rz 65 deg; joints [9.331, -43.934, 127.204, 74.433, -88.186, -6.482]
  MoveL 257 to (825.92, 1304.75, 0) mm, rotated rx 0 ry 90 rz 65 deg; joints [7.864, -45.069, 131.496, 72.895, -88.948, -3.415]
  MoveL 258 to (980.11, 1304.75, 0) mm, rotated rx 0 ry 90 rz 65 deg; joints [6.933, -41.57, 119.511, 72.307, -86.285, -11.481]
  MoveL 259 to (1047.26, 1203.15, 0) mm, rotated rx 0 ry 90 rz 65 deg; joints [10.784, -39.2, 112.664, 76.35, -85.992, -16.055]
  MoveL 260 to (998.73, 1203.15, 0) mm, rotated rx 0 ry 90 rz 65 deg; joints [11.174, -40.616, 116.68, 76.566, -86.701, -13.547]
  MoveL 261 to (964.84, 1254.43, 0) mm, rotated rx 0 ry 90 rz 65 deg; joints [9.233, -41.785, 120.165, 74.54, -86.863, -11.194]
  MoveL 262 to (962.71, 1257.22, 0) mm, rotated rx 0 ry 90 rz 65 deg; joints [9.126, -41.852, 120.371, 74.428, -86.879, -11.054]
  MoveL 263 to (960.25, 1259.66, 0) mm, rotated rx 0 ry 90 rz 65 deg; joints [9.035, -41.926, 120.599, 74.331, -86.903, -10.901]
  MoveL 264 to (957.52, 1261.76, 0) mm, rotated rx 0 ry 90 rz 65 deg; joints [8.962, -42.005, 120.844, 74.25, -86.934, -10.737]
  MoveL 265 to (954.55, 1263.49, 0) mm, rotated rx 0 ry 90 rz 65 deg; joints [8.906, -42.089, 121.103, 74.186, -86.972, -10.565]
  MoveL 266 to (951.38, 1264.86, 0) mm, rotated rx 0 ry 90 rz 65 deg; joints [8.867, -42.175, 121.371, 74.139, -87.015, -10.388]
  MoveL 267 to (948.07, 1265.85, 0) mm, rotated rx 0 ry 90 rz 65 deg; joints [8.847, -42.263, 121.646, 74.109, -87.062, -10.206]
  MoveL 268 to (941.19, 1266.65, 0) mm, rotated rx 0 ry 90 rz 65 deg; joints [8.859, -42.438, 122.201, 74.102, -87.168, -9.841]
  MoveL 269 to (892.95, 1266.65, 0) mm, rotated rx 0 ry 90 rz 65 deg; joints [9.208, -43.581, 125.97, 74.34, -87.934, -7.327]
  MoveL 270 to (1053.1, 1149.78, 0) mm, rotated rx 0 ry 90 rz 65 deg; joints [12.889, -38.678, 111.232, 78.431, -86.394, -17.081]
  Set speed (60.0 mm/s)
  MoveL 271 to (898.67, 1149.78, 0) mm, rotated rx 0 ry 90 rz 65 deg; joints [14.471, -42.885, 123.639, 79.605, -88.318, -9.093]
  MoveL 272 to (894.63, 1149.99, 0) mm, rotated rx 0 ry 90 rz 65 deg; joints [14.508, -42.98, 123.952, 79.635, -88.363, -8.88]
  MoveL 273 to (890.72, 1150.63, 0) mm, rotated rx 0 ry 90 rz 65 deg; joints [14.525, -43.075, 124.265, 79.646, -88.404, -8.666]
  MoveL 274 to (886.94, 1151.67, 0) mm, rotated rx 0 ry 90 rz 65 deg; joints [14.522, -43.168, 124.574, 79.637, -88.443, -8.453]
  MoveL 275 to (883.33, 1153.13, 0) mm, rotated rx 0 ry 90 rz 65 deg; joints [14.499, -43.259, 124.878, 79.608, -88.478, -8.243]
  MoveL 276 to (879.91, 1154.97, 0) mm, rotated rx 0 ry 90 rz 65 deg; joints [14.455, -43.348, 125.175, 79.56, -88.509, -8.037]
  MoveL 277 to (876.69, 1157.21, 0) mm, rotated rx 0 ry 90 rz 65 deg; joints [14.391, -43.433, 125.463, 79.491, -88.537, -7.835]
  MoveL 278 to (873.71, 1159.83, 0) mm, rotated rx 0 ry 90 rz 65 deg; joints [14.307, -43.514, 125.74, 79.403, -88.562, -7.641]
  MoveL 279 to (870.99, 1162.83, 0) mm, rotated rx 0 ry 90 rz 65 deg; joints [14.202, -43.591, 126.004, 79.294, -88.583, -7.454]
  MoveL 280 to (868.67, 1166, 0) mm, rotated rx 0 ry 90 rz 65 deg; joints [14.084, -43.659, 126.24, 79.173, -88.599, -7.286]
  MoveL 281 to (866.69, 1169.36, 0) mm, rotated rx 0 ry 90 rz 65 deg; joints [13.952, -43.721, 126.453, 79.039, -88.611, -7.134]
  MoveL 282 to (865.04, 1172.89, 0) mm, rotated rx 0 ry 90 rz 65 deg; joints [13.809, -43.775, 126.644, 78.894, -88.619, -6.997]
  MoveL 283 to (863.72, 1176.55, 0) mm, rotated rx 0 ry 90 rz 65 deg; joints [13.656, -43.823, 126.811, 78.738, -88.624, -6.876]
  MoveL 284 to (862.71, 1180.31, 0) mm, rotated rx 0 ry 90 rz 65 deg; joints [13.493, -43.864, 126.956, 78.575, -88.625, -6.77]
  MoveL 285 to (862, 1184.14, 0) mm, rotated rx 0 ry 90 rz 65 deg; joints [13.324, -43.899, 127.079, 78.404, -88.623, -6.68]
  MoveL 286 to (861.58, 1188.01, 0) mm, rotated rx 0 ry 90 rz 65 deg; joints [13.149, -43.927, 127.179, 78.228, -88.617, -6.605]
  MoveL 287 to (861.44, 1191.9, 0) mm, rotated rx 0 ry 90 rz 65 deg; joints [12.97, -43.949, 127.257, 78.049, -88.608, -6.546]
  MoveL 288 to (861.44, 1246.06, 0) mm, rotated rx 0 ry 90 rz 65 deg; joints [10.429, -44.185, 128.107, 75.507, -88.473, -5.884]
  MoveL 289 to (823.34, 1246.06, 0) mm, rotated rx 0 ry 90 rz 65 deg; joints [10.772, -44.939, 130.97, 75.804, -89.025, -3.847]
  MoveL 290 to (823.34, 1108.29, 0) mm, rotated rx 0 ry 90 rz 65 deg; joints [17.321, -44.269, 128.412, 82.36, -89.219, -5.805]
  MoveL 291 to (1061.99, 1108.29, 0) mm, rotated rx 0 ry 90 rz 65 deg; joints [14.445, -38.085, 109.627, 79.977, -86.675, -18.166]
  MoveL 292 to (1059.69, 1118.65, 0) mm, rotated rx 0 ry 90 rz 65 deg; joints [14.061, -38.24, 110.044, 79.596, -86.603, -17.887]
  MoveL 293 to (1053.1, 1149.78, 0) mm, rotated rx 0 ry 90 rz 65 deg; joints [12.889, -38.678, 111.232, 78.431, -86.394, -17.081]
  MoveL 294 to (824.97, 1409.86, 0) mm, rotated rx 0 ry 90 rz 65 deg; joints [2.61, -45.262, 132.291, 67.637, -88.869, -2.747]
  Set speed (60.0 mm/s)
  MoveL 295 to (822.36, 1409.74, 0) mm, rotated rx 0 ry 90 rz 65 deg; joints [2.622, -45.309, 132.488, 67.646, -88.926, -2.609]
  MoveL 296 to (819.76, 1409.4, 0) mm, rotated rx 0 ry 90 rz 65 deg; joints [2.645, -45.354, 132.681, 67.667, -88.984, -2.473]
  MoveL 297 to (817.21, 1408.83, 0) mm, rotated rx 0 ry 90 rz 65 deg; joints [2.68, -45.398, 132.87, 67.699, -89.04, -2.339]
  MoveL 298 to (814.73, 1408.05, 0) mm, rotated rx 0 ry 90 rz 65 deg; joints [2.726, -45.441, 133.053, 67.743, -89.095, -2.21]
  MoveL 299 to (812.32, 1407.04, 0) mm, rotated rx 0 ry 90 rz 65 deg; joints [2.783, -45.481, 133.229, 67.798, -89.149, -2.085]
  MoveL 300 to (810.02, 1405.82, 0) mm, rotated rx 0 ry 90 rz 65 deg; joints [2.851, -45.52, 133.397, 67.865, -89.2, -1.966]
  MoveL 301 to (807.83, 1404.39, 0) mm, rotated rx 0 ry 90 rz 65 deg; joints [2.93, -45.555, 133.555, 67.942, -89.248, -1.854]
  MoveL 302 to (805.78, 1402.74, 0) mm, rotated rx 0 ry 90 rz 65 deg; joints [3.019, -45.588, 133.701, 68.03, -89.294, -1.75]
  MoveL 303 to (803.9, 1400.91, 0) mm, rotated rx 0 ry 90 rz 65 deg; joints [3.119, -45.618, 133.833, 68.128, -89.335, -1.656]
  MoveL 304 to (802.24, 1398.91, 0) mm, rotated rx 0 ry 90 rz 65 deg; joints [3.226, -45.644, 133.949, 68.234, -89.372, -1.573]
  MoveL 305 to (800.79, 1396.77, 0) mm, rotated rx 0 ry 90 rz 65 deg; joints [3.34, -45.665, 134.048, 68.348, -89.403, -1.503]
  MoveL 306 to (799.57, 1394.51, 0) mm, rotated rx 0 ry 90 rz 65 deg; joints [3.46, -45.683, 134.128, 68.468, -89.429, -1.446]
  MoveL 307 to (798.61, 1392.12, 0) mm, rotated rx 0 ry 90 rz 65 deg; joints [3.586, -45.696, 134.189, 68.593, -89.45, -1.403]
  MoveL 308 to (797.9, 1389.64, 0) mm, rotated rx 0 ry 90 rz 65 deg; joints [3.716, -45.705, 134.23, 68.723, -89.464, -1.375]
  MoveL 309 to (797.46, 1387.08, 0) mm, rotated rx 0 ry 90 rz 65 deg; joints [3.85, -45.71, 134.249, 68.856, -89.473, -1.362]
  MoveL 310 to (797.32, 1384.46, 0) mm, rotated rx 0 ry 90 rz 65 deg; joints [3.986, -45.709, 134.247, 68.992, -89.476, -1.365]
  MoveL 311 to (797.32, 1108.32, 0) mm, rotated rx 0 ry 90 rz 65 deg; joints [17.702, -44.772, 130.312, 82.724, -89.434, -4.424]
  MoveL 312 to (746.36, 1146.42, 0) mm, rotated rx 0 ry 90 rz 65 deg; joints [16.62, -45.831, 134.812, 81.621, -89.851, -1.008]
  MoveL 313 to (746.36, 1447.96, 0) mm, rotated rx 0 ry 90 rz 65 deg; joints [0.739, -46.478, 138.183, 65.748, -90.7, 1.554]
  MoveL 314 to (912.14, 1447.96, 0) mm, rotated rx 0 ry 90 rz 65 deg; joints [0.638, -43.499, 125.69, 65.838, -86.787, -7.121]
  MoveL 315 to (979.29, 1346.36, 0) mm, rotated rx 0 ry 90 rz 65 deg; joints [5.109, -41.709, 119.932, 70.495, -86.018, -11.092]
  MoveL 316 to (930.76, 1346.36, 0) mm, rotated rx 0 ry 90 rz 65 deg; joints [5.307, -42.937, 123.809, 70.538, -86.936, -8.602]
  MoveL 317 to (896.87, 1397.63, 0) mm, rotated rx 0 ry 90 rz 65 deg; joints [3.034, -43.807, 126.755, 68.184, -87.368, -6.544]
  MoveL 318 to (894.74, 1400.42, 0) mm, rotated rx 0 ry 90 rz 65 deg; joints [2.907, -43.857, 126.932, 68.053, -87.401, -6.421]
  MoveL 319 to (892.28, 1402.87, 0) mm, rotated rx 0 ry 90 rz 65 deg; joints [2.796, -43.914, 127.132, 67.937, -87.442, -6.283]
  MoveL 320 to (889.55, 1404.96, 0) mm, rotated rx 0 ry 90 rz 65 deg; joints [2.703, -43.976, 127.351, 67.837, -87.492, -6.133]
  MoveL 321 to (886.57, 1406.7, 0) mm, rotated rx 0 ry 90 rz 65 deg; joints [2.627, -44.042, 127.587, 67.754, -87.548, -5.972]
  MoveL 322 to (883.41, 1408.07, 0) mm, rotated rx 0 ry 90 rz 65 deg; joints [2.568, -44.111, 127.837, 67.689, -87.61, -5.803]
  MoveL 323 to (880.1, 1409.05, 0) mm, rotated rx 0 ry 90 rz 65 deg; joints [2.528, -44.182, 128.095, 67.642, -87.677, -5.628]
  MoveL 324 to (873.22, 1409.86, 0) mm, rotated rx 0 ry 90 rz 65 deg; joints [2.504, -44.327, 128.627, 67.604, -87.822, -5.269]
  MoveL 325 to (824.97, 1409.86, 0) mm, rotated rx 0 ry 90 rz 65 deg; joints [2.61, -45.262, 132.291, 67.637, -88.869, -2.747]
  MoveL 326 to (667.84, 1086.24, 0) mm, rotated rx 0 ry 90 rz 65 deg; joints [21.01, -46.587, 138.836, 86.013, -90.156, 2.244]
  Set speed (60.0 mm/s)
  MoveL 327 to (664.42, 1088.09, 0) mm, rotated rx 0 ry 90 rz 65 deg; joints [20.982, -46.632, 139.116, 85.986, -90.174, 2.478]
  MoveL 328 to (661.2, 1090.32, 0) mm, rotated rx 0 ry 90 rz 65 deg; joints [20.931, -46.675, 139.39, 85.935, -90.193, 2.709]
  MoveL 329 to (658.22, 1092.94, 0) mm, rotated rx 0 ry 90 rz 65 deg; joints [20.854, -46.715, 139.658, 85.859, -90.213, 2.935]
  MoveL 330 to (655.5, 1095.94, 0) mm, rotated rx 0 ry 90 rz 65 deg; joints [20.752, -46.754, 139.918, 85.759, -90.234, 3.156]
  MoveL 331 to (653.18, 1099.11, 0) mm, rotated rx 0 ry 90 rz 65 deg; joints [20.633, -46.788, 140.155, 85.641, -90.256, 3.357]
  MoveL 332 to (651.2, 1102.47, 0) mm, rotated rx 0 ry 90 rz 65 deg; joints [20.496, -46.818, 140.373, 85.505, -90.279, 3.543]
  MoveL 333 to (649.55, 1106, 0) mm, rotated rx 0 ry 90 rz 65 deg; joints [20.343, -46.846, 140.572, 85.353, -90.302, 3.713]
  MoveL 334 to (648.23, 1109.66, 0) mm, rotated rx 0 ry 90 rz 65 deg; joints [20.177, -46.87, 140.751, 85.188, -90.326, 3.868]
  MoveL 335 to (647.22, 1113.42, 0) mm, rotated rx 0 ry 90 rz 65 deg; joints [19.998, -46.891, 140.912, 85.01, -90.35, 4.005]
  MoveL 336 to (646.51, 1117.25, 0) mm, rotated rx 0 ry 90 rz 65 deg; joints [19.808, -46.909, 141.053, 84.822, -90.375, 4.126]
  MoveL 337 to (646.09, 1121.13, 0) mm, rotated rx 0 ry 90 rz 65 deg; joints [19.61, -46.925, 141.174, 84.625, -90.399, 4.231]
  MoveL 338 to (645.95, 1125.01, 0) mm, rotated rx 0 ry 90 rz 65 deg; joints [19.406, -46.938, 141.276, 84.422, -90.423, 4.318]
  MoveL 339 to (645.95, 1228.44, 0) mm, rotated rx 0 ry 90 rz 65 deg; joints [13.713, -47.16, 143.369, 78.778, -91.213, 6.09]
  MoveL 340 to (607.85, 1228.44, 0) mm, rotated rx 0 ry 90 rz 65 deg; joints [14.26, -47.32, 145.956, 79.379, -91.604, 8.487]
  MoveL 341 to (607.85, 1041.4, 0) mm, rotated rx 0 ry 90 rz 65 deg; joints [24.61, -46.972, 141.561, 89.611, -90.031, 4.589]
  MoveL 342 to (1071.45, 1041.4, 0) mm, rotated rx 0 ry 90 rz 65 deg; joints [16.923, -37.18, 107.224, 82.403, -87.251, -19.774]
  MoveL 343 to (1066.6, 1051.72, 0) mm, rotated rx 0 ry 90 rz 65 deg; joints [16.586, -37.437, 107.901, 82.064, -87.195, -19.341]
  MoveL 344 to (1052.59, 1082.89, 0) mm, rotated rx 0 ry 90 rz 65 deg; joints [15.537, -38.167, 109.847, 81.009, -87.038, -18.087]
  MoveL 345 to (683.18, 1082.89, 0) mm, rotated rx 0 ry 90 rz 65 deg; joints [20.881, -46.396, 137.709, 85.882, -90.094, 1.31]
  MoveL 346 to (679.15, 1083.11, 0) mm, rotated rx 0 ry 90 rz 65 deg; joints [20.948, -46.445, 137.989, 85.95, -90.109, 1.54]
  MoveL 347 to (675.23, 1083.74, 0) mm, rotated rx 0 ry 90 rz 65 deg; joints [20.992, -46.494, 138.271, 85.994, -90.124, 1.774]
  MoveL 348 to (671.45, 1084.79, 0) mm, rotated rx 0 ry 90 rz 65 deg; joints [21.013, -46.541, 138.554, 86.015, -90.14, 2.009]
  MoveL 349 to (667.84, 1086.24, 0) mm, rotated rx 0 ry 90 rz 65 deg; joints [21.01, -46.587, 138.836, 86.013, -90.156, 2.244]
  MoveL 350 to (819.97, 1615.51, 0) mm, rotated rx 0 ry 90 rz 65 deg; joints [-7.762, -45.185, 131.971, 57.279, -88.261, -2.704]
  Set speed (60.0 mm/s)
  MoveL 351 to (815.87, 1618.52, 0) mm, rotated rx 0 ry 90 rz 65 deg; joints [-7.94, -45.251, 132.245, 57.096, -88.366, -2.523]
  MoveL 352 to (811.76, 1620.83, 0) mm, rotated rx 0 ry 90 rz 65 deg; joints [-8.085, -45.318, 132.527, 56.946, -88.477, -2.339]
  MoveL 353 to (807.64, 1622.44, 0) mm, rotated rx 0 ry 90 rz 65 deg; joints [-8.195, -45.386, 132.817, 56.832, -88.594, -2.15]
  MoveL 354 to (803.51, 1623.35, 0) mm, rotated rx 0 ry 90 rz 65 deg; joints [-8.271, -45.454, 133.113, 56.751, -88.716, -1.958]
  MoveL 355 to (799.39, 1623.57, 0) mm, rotated rx 0 ry 90 rz 65 deg; joints [-8.312, -45.524, 133.415, 56.706, -88.842, -1.762]
  MoveL 356 to (795.28, 1623.11, 0) mm, rotated rx 0 ry 90 rz 65 deg; joints [-8.319, -45.593, 133.724, 56.695, -88.973, -1.562]
  MoveL 357 to (791.18, 1621.96, 0) mm, rotated rx 0 ry 90 rz 65 deg; joints [-8.292, -45.663, 134.038, 56.719, -89.108, -1.359]
  MoveL 358 to (787.11, 1620.15, 0) mm, rotated rx 0 ry 90 rz 65 deg; joints [-8.229, -45.733, 134.357, 56.778, -89.246, -1.151]
  MoveL 359 to (783.08, 1617.67, 0) mm, rotated rx 0 ry 90 rz 65 deg; joints [-8.132, -45.803, 134.68, 56.873, -89.386, -0.94]
  MoveL 360 to (779.07, 1614.52, 0) mm, rotated rx 0 ry 90 rz 65 deg; joints [-7.999, -45.872, 135.006, 57.004, -89.528, -0.726]
  MoveL 361 to (775.12, 1610.72, 0) mm, rotated rx 0 ry 90 rz 65 deg; joints [-7.831, -45.94, 135.334, 57.171, -89.672, -0.509]
  MoveL 362 to (767.37, 1601.17, 0) mm, rotated rx 0 ry 90 rz 65 deg; joints [-7.387, -46.074, 135.994, 57.613, -89.957, -0.067]
  MoveL 363 to (761.62, 1592.15, 0) mm, rotated rx 0 ry 90 rz 65 deg; joints [-6.951, -46.172, 136.496, 58.049, -90.171, 0.275]
  MoveL 364 to (756.45, 1582.48, 0) mm, rotated rx 0 ry 90 rz 65 deg; joints [-6.472, -46.259, 136.955, 58.53, -90.363, 0.593]
  MoveL 365 to (747.84, 1562.64, 0) mm, rotated rx 0 ry 90 rz 65 deg; joints [-5.461, -46.4, 137.731, 59.546, -90.675, 1.147]
  MoveL 366 to (740.38, 1540.88, 0) mm, rotated rx 0 ry 90 rz 65 deg; joints [-4.32, -46.516, 138.406, 60.693, -90.925, 1.648]
  MoveL 367 to (728.8, 1495.08, 0) mm, rotated rx 0 ry 90 rz 65 deg; joints [-1.849, -46.679, 139.422, 63.178, -91.238, 2.447]
  MoveL 368 to (721.23, 1451.76, 0) mm, rotated rx 0 ry 90 rz 65 deg; joints [0.545, -46.766, 140.002, 65.579, -91.339, 2.947]
  MoveL 369 to (714.36, 1388.82, 0) mm, rotated rx 0 ry 90 rz 65 deg; joints [4.064, -46.81, 140.314, 69.1, -91.251, 3.273]
  MoveL 370 to (711.2, 1304.56, 0) mm, rotated rx 0 ry 90 rz 65 deg; joints [8.745, -46.746, 139.864, 73.768, -90.872, 2.993]
  MoveL 371 to (711.2, 1115.64, 0) mm, rotated rx 0 ry 90 rz 65 deg; joints [18.723, -46.19, 136.593, 83.723, -90.044, 0.4]
  MoveL 372 to (673.1, 1115.64, 0) mm, rotated rx 0 ry 90 rz 65 deg; joints [19.396, -46.647, 139.214, 84.402, -90.251, 2.554]
  MoveL 373 to (673.1, 1968.88, 0) mm, rotated rx 0 ry 90 rz 65 deg; joints [-27.309, -45.768, 134.519, 37.698, -89.011, -0.764]
  MoveL 374 to (1130.3, 1335.87, 0) mm, rotated rx 0 ry 90 rz 65 deg; joints [4.99, -37.118, 107.061, 71.115, -83.261, -18.935]
  MoveL 375 to (1130.3, 1042.48, 0) mm, rotated rx 0 ry 90 rz 65 deg; joints [16.23, -35.195, 102.113, 81.922, -86.573, -22.84]
  MoveL 376 to (1092.2, 1121.07, 0) mm, rotated rx 0 ry 90 rz 65 deg; joints [13.654, -37.214, 107.312, 79.316, -86.16, -19.542]
  MoveL 377 to (1085.99, 1117.44, 0) mm, rotated rx 0 ry 90 rz 65 deg; joints [13.853, -37.388, 107.772, 79.485, -86.279, -19.274]
  MoveL 378 to (1081.58, 1154.26, 0) mm, rotated rx 0 ry 90 rz 65 deg; joints [12.458, -37.811, 108.893, 78.115, -85.963, -18.497]
  MoveL 379 to (1068.65, 1225.33, 0) mm, rotated rx 0 ry 90 rz 65 deg; joints [9.727, -38.664, 111.194, 75.401, -85.464, -16.889]
  MoveL 380 to (1058.35, 1263.64, 0) mm, rotated rx 0 ry 90 rz 65 deg; joints [8.234, -39.17, 112.584, 73.895, -85.276, -15.918]
  MoveL 381 to (1051.94, 1282.64, 0) mm, rotated rx 0 ry 90 rz 65 deg; joints [7.487, -39.445, 113.347, 73.134, -85.214, -15.388]
  MoveL 382 to (1044.63, 1300.77, 0) mm, rotated rx 0 ry 90 rz 65 deg; joints [6.772, -39.733, 114.154, 72.4, -85.181, -14.833]
  MoveL 383 to (1027.17, 1332.11, 0) mm, rotated rx 0 ry 90 rz 65 deg; joints [5.532, -40.345, 115.896, 71.104, -85.23, -13.655]
  MoveL 384 to (832.1, 1602.19, 0) mm, rotated rx 0 ry 90 rz 65 deg; joints [-7.023, -44.994, 131.192, 58.034, -87.985, -3.225]
  MoveL 385 to (824.05, 1611.79, 0) mm, rotated rx 0 ry 90 rz 65 deg; joints [-7.55, -45.12, 131.703, 57.497, -88.162, -2.881]
  MoveL 386 to (819.97, 1615.51, 0) mm, rotated rx 0 ry 90 rz 65 deg; joints [-7.762, -45.185, 131.971, 57.279, -88.261, -2.704]
  MoveL 387 to (1051.03, 1672.5, 0) mm, rotated rx 0 ry 90 rz 65 deg; joints [-8.813, -39.334, 113.038, 57.264, -81.016, -13.653]
  Set speed (60.0 mm/s)
  MoveL 388 to (1042.85, 1679.23, 0) mm, rotated rx 0 ry 90 rz 65 deg; joints [-9.144, -39.548, 113.635, 56.888, -81.148, -13.277]
  MoveL 389 to (1034.8, 1688.83, 0) mm, rotated rx 0 ry 90 rz 65 deg; joints [-9.596, -39.741, 114.176, 56.398, -81.237, -12.914]
  MoveL 390 to (839.73, 1958.92, 0) mm, rotated rx 0 ry 90 rz 65 deg; joints [-23.403, -42.775, 123.283, 41.99, -82.915, -6.335]
  MoveL 391 to (822.27, 1990.25, 0) mm, rotated rx 0 ry 90 rz 65 deg; joints [-25.04, -42.85, 123.526, 40.335, -82.866, -6.02]
  MoveL 392 to (814.96, 2008.38, 0) mm, rotated rx 0 ry 90 rz 65 deg; joints [-25.935, -42.821, 123.43, 39.444, -82.722, -5.95]
  MoveL 393 to (808.55, 2027.39, 0) mm, rotated rx 0 ry 90 rz 65 deg; joints [-26.844, -42.755, 123.216, 38.544, -82.513, -5.927]
  MoveL 394 to (798.26, 2065.69, 0) mm, rotated rx 0 ry 90 rz 65 deg; joints [-28.608, -42.539, 122.522, 36.813, -81.951, -5.983]
  MoveL 395 to (787.07, 2124.74, 0) mm, rotated rx 0 ry 90 rz 65 deg; joints [-31.166, -42.036, 120.938, 34.336, -80.799, -6.233]
  MoveL 396 to (778.57, 2199.46, 0) mm, rotated rx 0 ry 90 rz 65 deg; joints [-34.146, -41.145, 118.236, 31.504, -78.942, -6.704]
  MoveL 397 to (774.7, 2299.07, 0) mm, rotated rx 0 ry 90 rz 65 deg; joints [-37.686, -39.541, 113.614, 28.238, -75.888, -7.46]
  MoveL 398 to (774.7, 2323, 0) mm, rotated rx 0 ry 90 rz 65 deg; joints [-38.47, -39.087, 112.354, 27.533, -75.072, -7.648]
  MoveL 399 to (736.6, 2401.6, 0) mm, rotated rx 0 ry 90 rz 65 deg; joints [-41.945, -38.403, 110.485, 24.099, -73.555, -7.217]
  MoveL 400 to (736.6, 1955.16, 0) mm, rotated rx 0 ry 90 rz 65 deg; joints [-25.261, -44.871, 130.701, 39.814, -86.794, -2.669]
  MoveL 401 to (1193.8, 1322.14, 0) mm, rotated rx 0 ry 90 rz 65 deg; joints [5.299, -34.816, 101.16, 71.841, -82.226, -22.413]
  MoveL 402 to (1193.8, 2290.27, 0) mm, rotated rx 0 ry 90 rz 65 deg; joints [-28.867, -25.729, 79.58, 42.119, -61.548, -23.305]
  MoveL 403 to (1155.7, 2290.27, 0) mm, rotated rx 0 ry 90 rz 65 deg; joints [-29.493, -27.404, 83.414, 40.712, -62.929, -21.386]
  MoveL 404 to (1155.7, 1986.46, 0) mm, rotated rx 0 ry 90 rz 65 deg; joints [-19.711, -33.012, 96.692, 48.417, -71.824, -19.369]
  MoveL 405 to (1152.54, 1902.21, 0) mm, rotated rx 0 ry 90 rz 65 deg; joints [-16.773, -34.163, 99.528, 50.925, -73.878, -18.881]
  MoveL 406 to (1148.44, 1860.23, 0) mm, rotated rx 0 ry 90 rz 65 deg; joints [-15.294, -34.752, 100.998, 52.187, -74.9, -18.556]
  MoveL 407 to (1142.38, 1818.5, 0) mm, rotated rx 0 ry 90 rz 65 deg; joints [-13.813, -35.358, 102.526, 53.449, -75.924, -18.163]
  MoveL 408 to (1132.84, 1772.91, 0) mm, rotated rx 0 ry 90 rz 65 deg; joints [-12.182, -36.064, 104.325, 54.832, -77.066, -17.624]
  MoveL 409 to (1126.52, 1750.15, 0) mm, rotated rx 0 ry 90 rz 65 deg; joints [-11.363, -36.446, 105.311, 55.521, -77.656, -17.291]
  MoveL 410 to (1119.06, 1728.39, 0) mm, rotated rx 0 ry 90 rz 65 deg; joints [-10.58, -36.845, 106.346, 56.174, -78.243, -16.913]
  MoveL 411 to (1110.45, 1708.54, 0) mm, rotated rx 0 ry 90 rz 65 deg; joints [-9.867, -37.254, 107.419, 56.758, -78.815, -16.486]
  MoveL 412 to (1105.28, 1698.87, 0) mm, rotated rx 0 ry 90 rz 65 deg; joints [-9.522, -37.481, 108.017, 57.035, -79.115, -16.235]
  MoveL 413 to (1099.53, 1689.86, 0) mm, rotated rx 0 ry 90 rz 65 deg; joints [-9.204, -37.719, 108.648, 57.284, -79.416, -15.956]
  MoveL 414 to (1091.78, 1680.3, 0) mm, rotated rx 0 ry 90 rz 65 deg; joints [-8.873, -38.02, 109.453, 57.53, -79.777, -15.584]
  MoveL 415 to (1083.83, 1673.36, 0) mm, rotated rx 0 ry 90 rz 65 deg; joints [-8.643, -38.31, 110.232, 57.681, -80.101, -15.203]
  MoveL 416 to (1079.79, 1670.87, 0) mm, rotated rx 0 ry 90 rz 65 deg; joints [-8.568, -38.45, 110.612, 57.72, -80.248, -15.01]
  MoveL 417 to (1075.72, 1669.06, 0) mm, rotated rx 0 ry 90 rz 65 deg; joints [-8.52, -38.587, 110.984, 57.733, -80.386, -14.816]
  MoveL 418 to (1071.62, 1667.92, 0) mm, rotated rx 0 ry 90 rz 65 deg; joints [-8.498, -38.721, 111.349, 57.722, -80.515, -14.622]
  MoveL 419 to (1067.51, 1667.46, 0) mm, rotated rx 0 ry 90 rz 65 deg; joints [-8.504, -38.852, 111.706, 57.684, -80.634, -14.427]
  MoveL 420 to (1063.39, 1667.68, 0) mm, rotated rx 0 ry 90 rz 65 deg; joints [-8.538, -38.978, 112.054, 57.619, -80.744, -14.232]
  MoveL 421 to (1059.27, 1668.59, 0) mm, rotated rx 0 ry 90 rz 65 deg; joints [-8.601, -39.101, 112.392, 57.528, -80.845, -14.038]
  MoveL 422 to (1055.14, 1670.19, 0) mm, rotated rx 0 ry 90 rz 65 deg; joints [-8.693, -39.22, 112.72, 57.41, -80.935, -13.845]
  MoveL 423 to (1051.03, 1672.5, 0) mm, rotated rx 0 ry 90 rz 65 deg; joints [-8.813, -39.334, 113.038, 57.264, -81.016, -13.653]
  MoveL 424 to (152.4, 2122.08, 0) mm, rotated rx 0 ry 90 rz 65 deg; joints [-55.039, -46.321, 155.405, 10.528, -108.785, 3.425]
  Set speed (60.0 mm/s)
  MoveL 425 to (242.26, 2181.47, 0) mm, rotated rx 0 ry 90 rz 65 deg; joints [-52.536, -47.322, 148.672, 12.705, -101.079, 2.481]
  MoveL 426 to (245.1, 2183.49, 0) mm, rotated rx 0 ry 90 rz 65 deg; joints [-52.471, -47.329, 148.444, 12.761, -100.847, 2.44]
  MoveL 427 to (247.78, 2185.69, 0) mm, rotated rx 0 ry 90 rz 65 deg; joints [-52.422, -47.335, 148.213, 12.801, -100.614, 2.396]
  MoveL 428 to (250.31, 2188.06, 0) mm, rotated rx 0 ry 90 rz 65 deg; joints [-52.387, -47.339, 147.979, 12.826, -100.38, 2.349]
  MoveL 429 to (252.67, 2190.59, 0) mm, rotated rx 0 ry 90 rz 65 deg; joints [-52.367, -47.342, 147.743, 12.838, -100.146, 2.299]
  MoveL 430 to (254.87, 2193.27, 0) mm, rotated rx 0 ry 90 rz 65 deg; joints [-52.36, -47.344, 147.505, 12.835, -99.912, 2.246]
  MoveL 431 to (256.89, 2196.08, 0) mm, rotated rx 0 ry 90 rz 65 deg; joints [-52.367, -47.344, 147.267, 12.818, -99.68, 2.191]
  MoveL 432 to (258.73, 2199.02, 0) mm, rotated rx 0 ry 90 rz 65 deg; joints [-52.388, -47.343, 147.029, 12.789, -99.45, 2.134]
  MoveL 433 to (260.4, 2202.07, 0) mm, rotated rx 0 ry 90 rz 65 deg; joints [-52.421, -47.34, 146.791, 12.746, -99.223, 2.076]
  MoveL 434 to (261.87, 2205.21, 0) mm, rotated rx 0 ry 90 rz 65 deg; joints [-52.467, -47.336, 146.558, 12.692, -99, 2.018]
  MoveL 435 to (263.14, 2208.43, 0) mm, rotated rx 0 ry 90 rz 65 deg; joints [-52.525, -47.331, 146.327, 12.626, -98.783, 1.959]
  MoveL 436 to (264.23, 2211.71, 0) mm, rotated rx 0 ry 90 rz 65 deg; joints [-52.594, -47.324, 146.101, 12.549, -98.57, 1.9]
  MoveL 437 to (265.11, 2215.05, 0) mm, rotated rx 0 ry 90 rz 65 deg; joints [-52.674, -47.317, 145.88, 12.461, -98.364, 1.841]
  MoveL 438 to (265.81, 2218.43, 0) mm, rotated rx 0 ry 90 rz 65 deg; joints [-52.764, -47.309, 145.663, 12.363, -98.164, 1.783]
  MoveL 439 to (266.3, 2221.85, 0) mm, rotated rx 0 ry 90 rz 65 deg; joints [-52.865, -47.3, 145.453, 12.255, -97.97, 1.725]
  MoveL 440 to (266.6, 2225.3, 0) mm, rotated rx 0 ry 90 rz 65 deg; joints [-52.975, -47.29, 145.249, 12.138, -97.783, 1.668]
  MoveL 441 to (266.7, 2228.76, 0) mm, rotated rx 0 ry 90 rz 65 deg; joints [-53.095, -47.28, 145.052, 12.012, -97.604, 1.613]
  MoveL 442 to (266.7, 2374.4, 0) mm, rotated rx 0 ry 90 rz 65 deg; joints [-57.742, -46.165, 136.462, 7.258, -90.295, 0.038]
  MoveL 443 to (304.8, 2374.4, 0) mm, rotated rx 0 ry 90 rz 65 deg; joints [-56.064, -45.855, 134.928, 8.937, -89.084, -0.144]
  MoveL 444 to (304.8, 2174.27, 0) mm, rotated rx 0 ry 90 rz 65 deg; joints [-49.244, -47.331, 146.343, 15.943, -98.67, 2.466]
  MoveL 445 to (152.4, 2073.55, 0) mm, rotated rx 0 ry 90 rz 65 deg; joints [-52.96, -45.422, 157.927, 13, -111.984, 4.939]
  MoveL 446 to (152.4, 2122.08, 0) mm, rotated rx 0 ry 90 rz 65 deg; joints [-55.039, -46.321, 155.405, 10.528, -108.785, 3.425]
  MoveL 447 to (1113.37, 952.5, 0) mm, rotated rx 0 ry 90 rz 65 deg; joints [19.687, -34.762, 101.024, 85.134, -87.864, -23.648]
  Set speed (60.0 mm/s)
  MoveL 448 to (88.9, 952.5, 0) mm, rotated rx 90 ry 60 rz 155 deg; joints [46.463, -41.135, 154.306, 109.872, -81.722, -8.281]
  MoveL 449 to (88.9, 914.4, 0) mm, rotated rx 90 ry 70 rz 155 deg; joints [49.831, -43.409, 156.449, 113.065, -80.54, 1.106]
  MoveL 450 to (1091.34, 914.4, 0) mm, rotated rx 0 ry 90 rz 65 deg; joints [21.336, -35.034, 101.706, 86.635, -88.55, -23.285]
  MoveL 451 to (1096.93, 923.88, 0) mm, rotated rx 0 ry 90 rz 65 deg; joints [20.923, -34.967, 101.538, 86.258, -88.38, -23.376]
  MoveL 452 to (1113.37, 952.5, 0) mm, rotated rx 0 ry 90 rz 65 deg; joints [19.687, -34.762, 101.024, 85.134, -87.864, -23.648]
  MoveL 453 to (1113.37, 889, 0) mm, rotated rx 0 ry 90 rz 65 deg; joints [21.921, -33.903, 98.883, 87.209, -88.698, -24.989]
  Set speed (60.0 mm/s)
  MoveL 454 to (1097.33, 860.38, 0) mm, rotated rx 0 ry 90 rz 65 deg; joints [23.14, -34.052, 99.251, 88.311, -89.22, -24.789]
  MoveL 455 to (1091.87, 850.9, 0) mm, rotated rx 0 ry 90 rz 65 deg; joints [23.547, -34.1, 99.371, 88.68, -89.392, -24.722]
  MoveL 456 to (88.9, 850.9, 0) mm, rotated rx 90 ry 80 rz 155 deg; joints [54.605, -45.179, 156.96, 117.817, -79.437, 9.159]
  MoveL 457 to (88.9, 889, 0) mm, rotated rx 90 ry 70 rz 155 deg; joints [51.005, -43.903, 155.209, 114.442, -80.833, -0.683]
  MoveL 458 to (1113.37, 889, 0) mm, rotated rx 0 ry 90 rz 65 deg; joints [21.921, -33.903, 98.883, 87.209, -88.698, -24.989]
  MoveL 459 to (1113.37, 825.5, 0) mm, rotated rx 0 ry 90 rz 65 deg; joints [24.087, -32.925, 96.478, 89.182, -89.593, -26.444]
  Set speed (60.0 mm/s)
  MoveL 460 to (88.9, 825.5, 0) mm, rotated rx 90 ry 80 rz 155 deg; joints [55.658, -45.655, 155.624, 119.124, -79.971, 7.358]
  MoveL 461 to (88.9, 787.4, 0) mm, rotated rx 0 ry 90 rz 65 deg; joints [59.423, -45.839, 156.884, 122.603, -78.288, 17.609]
  MoveL 462 to (1092.4, 787.4, 0) mm, rotated rx 0 ry 90 rz 65 deg; joints [25.683, -33.044, 96.77, 90.613, -90.303, -26.273]
  MoveL 463 to (1097.73, 796.89, 0) mm, rotated rx 0 ry 90 rz 65 deg; joints [25.284, -33.015, 96.699, 90.254, -90.126, -26.316]
  MoveL 464 to (1113.37, 825.5, 0) mm, rotated rx 0 ry 90 rz 65 deg; joints [24.087, -32.925, 96.478, 89.182, -89.593, -26.444]
  MoveL 465 to (1113.37, 762, 0) mm, rotated rx 0 ry 90 rz 65 deg; joints [26.182, -31.82, 93.799, 91.044, -90.555, -28.015]
  Set speed (60.0 mm/s)
  MoveL 466 to (1098.13, 733.39, 0) mm, rotated rx 0 ry 90 rz 65 deg; joints [27.354, -31.85, 93.872, 92.079, -91.104, -27.958]
  MoveL 467 to (1092.95, 723.9, 0) mm, rotated rx 0 ry 90 rz 65 deg; joints [27.745, -31.858, 93.893, 92.425, -91.287, -27.939]
  MoveL 468 to (88.9, 723.9, 0) mm, rotated rx 0 ry 90 rz 65 deg; joints [61.631, -46.826, 153.283, 125.491, -80.268, 13.336]
  MoveL 469 to (88.9, 762, 0) mm, rotated rx 0 ry 90 rz 65 deg; joints [60.343, -46.304, 155.466, 123.817, -79.054, 15.826]
  MoveL 470 to (1113.37, 762, 0) mm, rotated rx 0 ry 90 rz 65 deg; joints [26.182, -31.82, 93.799, 91.044, -90.555, -28.015]
  MoveL 471 to (1113.37, 698.5, 0) mm, rotated rx 0 ry 90 rz 65 deg; joints [28.205, -30.58, 90.835, 92.783, -91.589, -29.706]
  Set speed (60.0 mm/s)
  MoveL 472 to (88.9, 698.5, 0) mm, rotated rx 0 ry 90 rz 65 deg; joints [62.435, -47.066, 151.792, 126.515, -81.111, 11.788]
  MoveL 473 to (88.9, 660.4, 0) mm, rotated rx 0 ry 90 rz 65 deg; joints [63.564, -47.283, 149.506, 127.925, -82.416, 9.614]
  MoveL 474 to (1093.5, 660.4, 0) mm, rotated rx 0 ry 90 rz 65 deg; joints [29.729, -30.533, 90.725, 94.106, -92.349, -29.724]
  MoveL 475 to (1098.54, 669.89, 0) mm, rotated rx 0 ry 90 rz 65 deg; joints [29.348, -30.546, 90.755, 93.776, -92.159, -29.719]
  MoveL 476 to (1113.37, 698.5, 0) mm, rotated rx 0 ry 90 rz 65 deg; joints [28.205, -30.58, 90.835, 92.783, -91.589, -29.706]
  MoveL 477 to (1113.37, 635, 0) mm, rotated rx 0 ry 90 rz 65 deg; joints [30.154, -29.194, 87.569, 94.392, -92.7, -31.521]
  Set speed (60.0 mm/s)
  MoveL 478 to (1098.95, 606.38, 0) mm, rotated rx 0 ry 90 rz 65 deg; joints [31.267, -29.092, 87.33, 95.334, -93.294, -31.608]
  MoveL 479 to (1094.06, 596.9, 0) mm, rotated rx 0 ry 90 rz 65 deg; joints [31.636, -29.056, 87.247, 95.647, -93.492, -31.637]
  MoveL 480 to (88.9, 596.9, 0) mm, rotated rx 0 ry 90 rz 65 deg; joints [65.265, -47.305, 145.57, 129.971, -84.669, 6.325]
  MoveL 481 to (88.9, 635, 0) mm, rotated rx 0 ry 90 rz 65 deg; joints [64.27, -47.34, 147.95, 128.787, -83.307, 8.252]
  MoveL 482 to (1113.37, 635, 0) mm, rotated rx 0 ry 90 rz 65 deg; joints [30.154, -29.194, 87.569, 94.392, -92.7, -31.521]
  MoveL 483 to (88.9, 317.5, 0) mm, rotated rx 0 ry 90 rz 65 deg; joints [70.803, -43.731, 126.488, 135.574, -95.186, -5.063]
  Set speed (60.0 mm/s)
  MoveL 484 to (88.9, 279.4, 0) mm, rotated rx 0 ry 90 rz 65 deg; joints [71.379, -42.89, 123.656, 136.005, -96.671, -6.4]
  MoveL 485 to (1098.24, 279.4, 0) mm, rotated rx 0 ry 90 rz 65 deg; joints [40.023, -18.514, 63.531, 100.749, -100.558, -43.986]
  MoveL 486 to (1102.05, 288.92, 0) mm, rotated rx 0 ry 90 rz 65 deg; joints [39.72, -18.732, 64.006, 100.573, -100.3, -43.77]
  MoveL 487 to (1113.37, 317.5, 0) mm, rotated rx 0 ry 90 rz 65 deg; joints [38.802, -19.358, 65.376, 100.025, -99.536, -43.144]
  MoveL 488 to (88.9, 317.5, 0) mm, rotated rx 0 ry 90 rz 65 deg; joints [70.803, -43.731, 126.488, 135.574, -95.186, -5.063]
  MoveL 489 to (88.9, 254, 0) mm, rotated rx 0 ry 90 rz 65 deg; joints [71.744, -42.29, 121.733, 136.256, -97.668, -7.278]
  Set speed (60.0 mm/s)
  MoveL 490 to (1113.37, 254, 0) mm, rotated rx 0 ry 90 rz 65 deg; joints [40.322, -16.509, 59.178, 100.52, -101.203, -46.297]
  MoveL 491 to (1102.52, 225.42, 0) mm, rotated rx 0 ry 90 rz 65 deg; joints [41.202, -15.711, 57.456, 100.949, -102.016, -47.1]
  MoveL 492 to (1098.88, 215.9, 0) mm, rotated rx 0 ry 90 rz 65 deg; joints [41.493, -15.432, 56.855, 101.083, -102.291, -47.381]
  MoveL 493 to (88.9, 215.9, 0) mm, rotated rx 0 ry 90 rz 65 deg; joints [72.267, -41.333, 118.795, 136.577, -99.175, -8.582]
  MoveL 494 to (88.9, 254, 0) mm, rotated rx 0 ry 90 rz 65 deg; joints [71.744, -42.29, 121.733, 136.256, -97.668, -7.278]
  MoveL 495 to (88.9, 190.5, 0) mm, rotated rx 0 ry 90 rz 65 deg; joints [72.6, -40.657, 116.799, 136.756, -100.188, -9.445]
  Set speed (60.0 mm/s)
  MoveL 496 to (88.9, 152.4, 0) mm, rotated rx 0 ry 90 rz 65 deg; joints [73.077, -39.587, 113.743, 136.972, -101.72, -10.737]
  MoveL 497 to (1099.53, 152.4, 0) mm, rotated rx 0 ry 90 rz 65 deg; joints [42.897, -11.701, 48.88, 101.043, -104.173, -51.445]
  MoveL 498 to (1102.99, 161.93, 0) mm, rotated rx 0 ry 90 rz 65 deg; joints [42.619, -12.073, 49.668, 100.965, -103.876, -51.066]
  MoveL 499 to (1113.37, 190.5, 0) mm, rotated rx 0 ry 90 rz 65 deg; joints [41.776, -13.12, 51.9, 100.692, -103.003, -49.999]
  MoveL 500 to (88.9, 190.5, 0) mm, rotated rx 0 ry 90 rz 65 deg; joints [72.6, -40.657, 116.799, 136.756, -100.188, -9.445]
  MoveL 501 to (88.9, 127, 0) mm, rotated rx 0 ry 90 rz 65 deg; joints [73.381, -38.836, 111.664, 137.081, -102.752, -11.599]
  Set speed (60.0 mm/s)
  MoveL 502 to (1113.37, 127, 0) mm, rotated rx 0 ry 90 rz 65 deg; joints [43.167, -8.85, 42.854, 100.399, -104.98, -54.625]
  MoveL 503 to (1104.01, 98.53, 0) mm, rotated rx 0 ry 90 rz 65 deg; joints [43.96, -7.315, 39.631, 100.407, -105.937, -56.223]
  MoveL 504 to (1100.86, 88.9, 0) mm, rotated rx 0 ry 90 rz 65 deg; joints [44.225, -6.742, 38.433, 100.381, -106.271, -56.821]
  MoveL 505 to (88.9, 88.9, 0) mm, rotated rx 0 ry 90 rz 65 deg; joints [73.818, -37.654, 108.475, 137.191, -104.315, -12.9]
  MoveL 506 to (88.9, 127, 0) mm, rotated rx 0 ry 90 rz 65 deg; joints [73.381, -38.836, 111.664, 137.081, -102.752, -11.599]
  MoveL 507 to (88.9, 63.5, 0) mm, rotated rx 0 ry 90 rz 65 deg; joints [74.097, -36.827, 106.3, 137.229, -105.368, -13.775]
  Set speed (60.0 mm/s)
  MoveL 508 to (88.9, 25.4, 0) mm, rotated rx 0 ry 90 rz 65 deg; joints [74.498, -35.528, 102.958, 137.232, -106.969, -15.107]
  MoveL 509 to (1101.55, 25.4, 0) mm, rotated rx 0 ry 90 rz 65 deg; joints [45.507, 2.128, 20.105, 98.055, -108.922, -66.423]
  MoveL 510 to (1104.5, 35.01, 0) mm, rotated rx 0 ry 90 rz 65 deg; joints [45.255, 0.579, 23.276, 98.488, -108.458, -64.764]
  MoveL 511 to (1113.37, 63.5, 0) mm, rotated rx 0 ry 90 rz 65 deg; joints [44.498, -2.581, 29.782, 99.194, -107.269, -61.4]
  MoveL 512 to (88.9, 63.5, 0) mm, rotated rx 0 ry 90 rz 65 deg; joints [74.097, -36.827, 106.3, 137.229, -105.368, -13.775]
  MoveL 513 to (181.97, 1023.42, 0) mm, rotated rx 90 ry 70 rz 155 deg; joints [39.244, -43.118, 157.087, 103.06, -84.263, 3.312]
  Set speed (60.0 mm/s)
  MoveL 514 to (213.62, 1020.12, 0) mm, rotated rx 90 ry 70 rz 155 deg; joints [37.988, -43.834, 155.397, 102.107, -85.262, 1.06]
  MoveL 515 to (309.51, 1016, 0) mm, rotated rx 90 ry 80 rz 155 deg; joints [34.985, -46.026, 154.327, 99.489, -86.879, 8.042]
  MoveL 516 to (1130.3, 1016, 0) mm, rotated rx 0 ry 90 rz 65 deg; joints [17.196, -34.913, 101.402, 82.837, -86.895, -23.317]
  MoveL 517 to (1130.3, 977.9, 0) mm, rotated rx 0 ry 90 rz 65 deg; joints [18.569, -34.473, 100.3, 84.129, -87.371, -24.038]
  MoveL 518 to (105.83, 977.9, 0) mm, rotated rx 90 ry 60 rz 155 deg; joints [44.316, -40.968, 154.693, 107.791, -82.352, -7.474]
  MoveL 519 to (114.82, 1019.86, 0) mm, rotated rx 90 ry 60 rz 155 deg; joints [41.623, -40.305, 156.052, 105.051, -82.862, -5.197]
  MoveL 520 to (117.51, 1033.91, 0) mm, rotated rx 90 ry 60 rz 155 deg; joints [40.703, -40.063, 156.493, 104.131, -83.081, -4.429]
  MoveL 521 to (181.97, 1023.42, 0) mm, rotated rx 90 ry 70 rz 155 deg; joints [39.244, -43.118, 157.087, 103.06, -84.263, 3.312]
  MoveL 522 to (127, 1111.75, 0) mm, rotated rx 90 ry 50 rz 155 deg; joints [34.885, -36.502, 154.783, 98.724, -85.335, -12.075]
  Set speed (60.0 mm/s)
  MoveL 523 to (130.87, 2230.12, 0) mm, rotated rx 90 ry 10 rz 155 deg; joints [-40.156, -23.049, 134.121, 26.389, -109.042, -70.805]
  MoveL 524 to (135.96, 2280.2, 0) mm, rotated rx 0 ry 90 rz 65 deg; joints [-61.451, -47.342, 146.959, 3.599, -99.598, 0.601]
  MoveL 525 to (143.38, 2329.01, 0) mm, rotated rx 0 ry 90 rz 65 deg; joints [-62.435, -47.19, 143.714, 2.582, -96.518, 0.293]
  MoveL 526 to (148.96, 2356.87, 0) mm, rotated rx 0 ry 90 rz 65 deg; joints [-62.888, -46.998, 141.782, 2.12, -94.78, 0.177]
  MoveL 527 to (156.55, 2387.57, 0) mm, rotated rx 0 ry 90 rz 65 deg; joints [-63.287, -46.703, 139.575, 1.715, -92.871, 0.086]
  MoveL 528 to (153.12, 2391.32, 0) mm, rotated rx 0 ry 90 rz 65 deg; joints [-63.549, -46.683, 139.444, 1.452, -92.76, 0.07]
  MoveL 529 to (142.88, 2402.6, 0) mm, rotated rx 0 ry 90 rz 65 deg; joints [-64.329, -46.619, 139.037, 0.672, -92.417, 0.028]
  MoveL 530 to (136.31, 2403.48, 0) mm, rotated rx 0 ry 90 rz 65 deg; joints [-64.675, -46.643, 139.184, 0.325, -92.541, 0.014]
  MoveL 531 to (116.61, 2406.19, 0) mm, rotated rx 0 ry 90 rz 65 deg; joints [-65.724, -46.707, 139.603, -0.725, -92.896, -0.037]
  MoveL 532 to (116.73, 2405.9, 0) mm, rotated rx 0 ry 90 rz 65 deg; joints [-65.711, -46.709, 139.618, -0.712, -92.909, -0.036]
  MoveL 533 to (109.88, 2396.61, 0) mm, rotated rx 0 ry 90 rz 65 deg; joints [-65.847, -46.826, 140.429, -0.848, -93.603, -0.053]
  MoveL 534 to (88.9, 2369.07, 0) mm, rotated rx 0 ry 90 rz 65 deg; joints [-66.302, -47.11, 142.829, -1.308, -95.717, -0.13]
  MoveL 535 to (88.9, 1033.15, 0) mm, rotated rx 90 ry -40 rz 155 deg; joints [40.292, 0.858, 125.243, 102.457, -81.06, -94.877]
  MoveL 536 to (127, 1111.75, 0) mm, rotated rx 90 ry 50 rz 155 deg; joints [34.885, -36.502, 154.783, 98.724, -85.335, -12.075]
  MoveL 537 to (1152.9, 2384.87, 0) mm, rotated rx 0 ry 90 rz 65 deg; joints [-32.268, -25.051, 78.042, 38.832, -59.578, -22.175]
  Set speed (60.0 mm/s)
  MoveL 538 to (1152.9, 2346.77, 0) mm, rotated rx 0 ry 90 rz 65 deg; joints [-31.188, -26.097, 80.418, 39.506, -61.014, -21.779]
  MoveL 539 to (916.39, 2346.77, 0) mm, rotated rx 0 ry 90 rz 65 deg; joints [-35.834, -34.729, 100.939, 31.38, -69.376, -12.125]
  MoveL 540 to (911.15, 2346.54, 0) mm, rotated rx 0 ry 90 rz 65 deg; joints [-35.944, -34.892, 101.35, 31.217, -69.565, -11.947]
  MoveL 541 to (905.96, 2345.86, 0) mm, rotated rx 0 ry 90 rz 65 deg; joints [-36.039, -35.063, 101.781, 31.068, -69.767, -11.77]
  MoveL 542 to (900.87, 2344.73, 0) mm, rotated rx 0 ry 90 rz 65 deg; joints [-36.119, -35.24, 102.227, 30.934, -69.982, -11.594]
  MoveL 543 to (895.89, 2343.16, 0) mm, rotated rx 0 ry 90 rz 65 deg; joints [-36.182, -35.421, 102.686, 30.816, -70.207, -11.419]
  MoveL 544 to (891.08, 2341.15, 0) mm, rotated rx 0 ry 90 rz 65 deg; joints [-36.229, -35.606, 103.154, 30.716, -70.443, -11.249]
  MoveL 545 to (886.47, 2338.7, 0) mm, rotated rx 0 ry 90 rz 65 deg; joints [-36.258, -35.792, 103.63, 30.633, -70.685, -11.082]
  MoveL 546 to (882.1, 2335.83, 0) mm, rotated rx 0 ry 90 rz 65 deg; joints [-36.269, -35.979, 104.109, 30.57, -70.935, -10.921]
  MoveL 547 to (877.99, 2332.54, 0) mm, rotated rx 0 ry 90 rz 65 deg; joints [-36.26, -36.166, 104.589, 30.529, -71.189, -10.767]
  MoveL 548 to (874.24, 2328.88, 0) mm, rotated rx 0 ry 90 rz 65 deg; joints [-36.231, -36.35, 105.061, 30.509, -71.443, -10.621]
  MoveL 549 to (870.91, 2324.89, 0) mm, rotated rx 0 ry 90 rz 65 deg; joints [-36.182, -36.526, 105.519, 30.512, -71.694, -10.487]
  MoveL 550 to (868.01, 2320.61, 0) mm, rotated rx 0 ry 90 rz 65 deg; joints [-36.114, -36.696, 105.958, 30.538, -71.939, -10.365]
  MoveL 551 to (865.58, 2316.07, 0) mm, rotated rx 0 ry 90 rz 65 deg; joints [-36.026, -36.856, 106.375, 30.587, -72.176, -10.256]
  MoveL 552 to (863.65, 2311.31, 0) mm, rotated rx 0 ry 90 rz 65 deg; joints [-35.918, -37.005, 106.766, 30.658, -72.403, -10.16]
  MoveL 553 to (862.23, 2306.35, 0) mm, rotated rx 0 ry 90 rz 65 deg; joints [-35.792, -37.144, 107.129, 30.753, -72.617, -10.079]
  MoveL 554 to (861.36, 2301.23, 0) mm, rotated rx 0 ry 90 rz 65 deg; joints [-35.647, -37.269, 107.458, 30.87, -72.818, -10.014]
  MoveL 555 to (861.07, 2295.97, 0) mm, rotated rx 0 ry 90 rz 65 deg; joints [-35.484, -37.38, 107.751, 31.009, -73.002, -9.966]
  MoveL 556 to (861.07, 2101.89, 0) mm, rotated rx 0 ry 90 rz 65 deg; joints [-28.681, -40.595, 116.617, 37.145, -78.778, -8.386]
  MoveL 557 to (823.03, 2146.01, 0) mm, rotated rx 0 ry 90 rz 65 deg; joints [-31.148, -40.905, 117.526, 34.585, -78.92, -7.548]
  MoveL 558 to (810.12, 2160.48, 0) mm, rotated rx 0 ry 90 rz 65 deg; joints [-31.976, -41.002, 117.809, 33.728, -78.969, -7.28]
  MoveL 559 to (810.12, 2384.87, 0) mm, rotated rx 0 ry 90 rz 65 deg; joints [-39.513, -36.914, 106.528, 26.956, -71.673, -9.085]
  MoveL 560 to (1152.9, 2384.87, 0) mm, rotated rx 0 ry 90 rz 65 deg; joints [-32.268, -25.051, 78.042, 38.832, -59.578, -22.175]
  MoveL 561 to (1130.3, 2071.98, 0) mm, rotated rx 0 ry 90 rz 65 deg; joints [-22.976, -32.712, 95.959, 45.262, -70.464, -18.648]
  Set speed (60.0 mm/s)
  MoveL 562 to (1130.3, 2321.37, 0) mm, rotated rx 0 ry 90 rz 65 deg; joints [-30.846, -27.712, 84.124, 39.16, -62.755, -20.447]
  MoveL 563 to (941.34, 2321.37, 0) mm, rotated rx 0 ry 90 rz 65 deg; joints [-34.505, -34.512, 100.396, 32.831, -69.386, -12.798]
  MoveL 564 to (927.78, 2308.5, 0) mm, rotated rx 0 ry 90 rz 65 deg; joints [-34.393, -35.201, 102.128, 32.741, -70.287, -12.237]
  MoveL 565 to (886.51, 2270.42, 0) mm, rotated rx 0 ry 90 rz 65 deg; joints [-34.072, -37.167, 107.189, 32.518, -72.958, -10.583]
  MoveL 566 to (1041.4, 2270.42, 0) mm, rotated rx 0 ry 90 rz 65 deg; joints [-30.912, -32.276, 94.9, 37.31, -67.616, -16.183]
  MoveL 567 to (1046.65, 2270.12, 0) mm, rotated rx 0 ry 90 rz 65 deg; joints [-30.805, -32.096, 94.465, 37.486, -67.443, -16.393]
  MoveL 568 to (1051.78, 2269.25, 0) mm, rotated rx 0 ry 90 rz 65 deg; joints [-30.683, -31.932, 94.069, 37.671, -67.294, -16.596]
  MoveL 569 to (1056.74, 2267.84, 0) mm, rotated rx 0 ry 90 rz 65 deg; joints [-30.548, -31.784, 93.712, 37.866, -67.168, -16.788]
  MoveL 570 to (1061.5, 2265.9, 0) mm, rotated rx 0 ry 90 rz 65 deg; joints [-30.4, -31.653, 93.397, 38.066, -67.066, -16.971]
  MoveL 571 to (1066.04, 2263.47, 0) mm, rotated rx 0 ry 90 rz 65 deg; joints [-30.242, -31.539, 93.125, 38.272, -66.987, -17.142]
  MoveL 572 to (1070.32, 2260.58, 0) mm, rotated rx 0 ry 90 rz 65 deg; joints [-30.075, -31.444, 92.898, 38.481, -66.933, -17.299]
  MoveL 573 to (1074.31, 2257.24, 0) mm, rotated rx 0 ry 90 rz 65 deg; joints [-29.9, -31.368, 92.716, 38.691, -66.902, -17.442]
  MoveL 574 to (1077.97, 2253.49, 0) mm, rotated rx 0 ry 90 rz 65 deg; joints [-29.718, -31.312, 92.582, 38.901, -66.896, -17.569]
  MoveL 575 to (1081.26, 2249.39, 0) mm, rotated rx 0 ry 90 rz 65 deg; joints [-29.532, -31.277, 92.497, 39.107, -66.914, -17.679]
  MoveL 576 to (1084.13, 2245.02, 0) mm, rotated rx 0 ry 90 rz 65 deg; joints [-29.344, -31.262, 92.461, 39.306, -66.955, -17.769]
  MoveL 577 to (1086.57, 2240.41, 0) mm, rotated rx 0 ry 90 rz 65 deg; joints [-29.157, -31.267, 92.474, 39.498, -67.018, -17.84]
  MoveL 578 to (1088.59, 2235.59, 0) mm, rotated rx 0 ry 90 rz 65 deg; joints [-28.972, -31.292, 92.533, 39.68, -67.102, -17.891]
  MoveL 579 to (1090.16, 2230.62, 0) mm, rotated rx 0 ry 90 rz 65 deg; joints [-28.788, -31.336, 92.637, 39.853, -67.205, -17.922]
  MoveL 580 to (1091.29, 2225.52, 0) mm, rotated rx 0 ry 90 rz 65 deg; joints [-28.608, -31.397, 92.785, 40.016, -67.326, -17.934]
  MoveL 581 to (1091.97, 2220.34, 0) mm, rotated rx 0 ry 90 rz 65 deg; joints [-28.433, -31.477, 92.976, 40.167, -67.465, -17.926]
  MoveL 582 to (1092.2, 2215.1, 0) mm, rotated rx 0 ry 90 rz 65 deg; joints [-28.263, -31.573, 93.207, 40.306, -67.62, -17.898]
  MoveL 583 to (1092.2, 2071.98, 0) mm, rotated rx 0 ry 90 rz 65 deg; joints [-23.533, -34.092, 99.352, 44.216, -71.723, -16.969]
  MoveL 584 to (1130.3, 2071.98, 0) mm, rotated rx 0 ry 90 rz 65 deg; joints [-22.976, -32.712, 95.959, 45.262, -70.464, -18.648]
  MoveL 585 to (25.4, 25.4, 0) mm, rotated rx 0 ry 90 rz 65 deg; joints [76.876, -36.093, 104.4, 139.816, -106.905, -13.798]
  Set speed (60.0 mm/s)
  MoveL 586 to (25.4, 1049.87, 0) mm, rotated rx 90 ry 50 rz 155 deg; joints [43.43, -34.845, 157.098, 105.739, -80.287, -9.093]
  MoveL 587 to (53.9, 1041.51, 0) mm, rotated rx 90 ry 50 rz 155 deg; joints [42.41, -35.996, 155.564, 105.256, -81.509, -11.571]
  MoveL 588 to (63.5, 1038.74, 0) mm, rotated rx 90 ry 50 rz 155 deg; joints [42.079, -36.343, 155.037, 105.083, -81.894, -12.381]
  MoveL 589 to (63.5, 25.4, 0) mm, rotated rx 0 ry 90 rz 65 deg; joints [75.443, -35.767, 103.565, 138.263, -106.938, -14.57]
  MoveL 590 to (25.4, 25.4, 0) mm, rotated rx 0 ry 90 rz 65 deg; joints [76.876, -36.093, 104.4, 139.816, -106.905, -13.798]
  MoveL 591 to (63.5, 1197.57, 0) mm, rotated rx 90 ry 40 rz 155 deg; joints [31.569, -29.268, 156.273, 95.254, -86.052, -13.176]
  Set speed (60.0 mm/s)
  MoveL 592 to (63.5, 2361.36, 0) mm, rotated rx 90 ry 30.44 rz -25 deg; joints [-76.421, -19.361, 81.156, 167.089, -117.598, -65.622]
  MoveL 593 to (54.18, 2348.46, 0) mm, rotated rx -90 ry 60 rz -25 deg; joints [-77.59, -42.911, 142.354, 347.243, -99.214, -332.076]
  MoveL 594 to (25.4, 2310.32, 0) mm, rotated rx -90 ry 70 rz -25 deg; joints [-75.61, -45.256, 146.781, 349.176, -101.326, -342.15]
